  //---------------------------------------------------------------------------------------------------------------
  //---------------------------------------------------------------------------------------------------------------
  E_PROGRESS.PROGRESS_STARTUP:
    _InstanceCtrl[E_INSTANCE.BUFFER_OUTFEED_ROBOT].Cmd   := E_INSTANCE_CMD.DISABLE;
    //-----------------------------------------------------------------------------------
    CASE _InstanceState[E_INSTANCE.BUFFER_OUTFEED_ROBOT].State
    OF
      E_INSTANCE_STATE.DISABLED:
        CASE _InstanceState[E_INSTANCE.BUFFER_OUTFEED_ROBOT].Progress
        OF
          E_PROGRESS.PROGRESS_BUSY:           // check for startup to be done
          _eState                                 := E_PROGRESS.PROGRESS_CHECK; // go check next insatnce
        END_CASE
    END_CASE

  //---------------------------------------------------------------------------------------------------------------
  //---------------------------------------------------------------------------------------------------------------
  E_PROGRESS.PROGRESS_CHECK:
    _InstanceCtrl[E_INSTANCE.OUTFEED_ROBOT_R1].Cmd   := E_INSTANCE_CMD.DISABLE;
    //-----------------------------------------------------------------------------------
    CASE _InstanceState[E_INSTANCE.OUTFEED_ROBOT_R1].State
    OF
      E_INSTANCE_STATE.DISABLED:
        CASE _InstanceState[E_INSTANCE.OUTFEED_ROBOT_R1].Progress
        OF
          E_PROGRESS.PROGRESS_BUSY:           // check for startup to be done
          _eState                                 := E_PROGRESS.PROGRESS_OCCUPIED; // go check next insatnce
        END_CASE
    END_CASE

  //---------------------------------------------------------------------------------------------------------------
  //---------------------------------------------------------------------------------------------------------------
  E_PROGRESS.PROGRESS_OCCUPIED:
    _InstanceCtrl[E_INSTANCE.OUTFEED_ROBOT_R2].Cmd   := E_INSTANCE_CMD.DISABLE;
    //-----------------------------------------------------------------------------------
    CASE _InstanceState[E_INSTANCE.OUTFEED_ROBOT_R2].State
    OF
      E_INSTANCE_STATE.DISABLED:
        CASE _InstanceState[E_INSTANCE.OUTFEED_ROBOT_R2].Progress
        OF
          E_PROGRESS.PROGRESS_BUSY:           // check for startup to be done
          _eState                                 := E_PROGRESS.PROGRESS_WORKING; // go check next insatnce
        END_CASE
    END_CASE

  //---------------------------------------------------------------------------------------------------------------
  //---------------------------------------------------------------------------------------------------------------
  E_PROGRESS.PROGRESS_WORKING:
    _InstanceCtrl[E_INSTANCE.SENDER_FAST].Cmd     := E_INSTANCE_CMD.DISABLE;
    //-----------------------------------------------------------------------------------
    CASE _InstanceState[E_INSTANCE.SENDER_FAST].State
    OF
      E_INSTANCE_STATE.DISABLED:
        CASE _InstanceState[E_INSTANCE.SENDER_FAST].Progress
        OF
          E_PROGRESS.PROGRESS_BUSY:           // check for startup to be done
          _eState                                 := E_PROGRESS.PROGRESS_STILL_WORKING; // go check next insatnce
        END_CASE
    END_CASE

  //---------------------------------------------------------------------------------------------------------------
  //---------------------------------------------------------------------------------------------------------------
  E_PROGRESS.PROGRESS_STILL_WORKING:
    _InstanceCtrl[E_INSTANCE.SENDER_BUFFER_INFEED].Cmd   := E_INSTANCE_CMD.DISABLE;
    //-----------------------------------------------------------------------------------
    CASE _InstanceState[E_INSTANCE.SENDER_BUFFER_INFEED].State
    OF
      E_INSTANCE_STATE.DISABLED:
        CASE _InstanceState[E_INSTANCE.SENDER_BUFFER_INFEED].Progress
        OF
          E_PROGRESS.PROGRESS_BUSY:           // check for startup to be done
          _eState                                 := E_PROGRESS.PROGRESS_DONE;
        END_CASE
    END_CASE
END_CASE
//-----------------------------------------------------------------------------
//-----------------------------------------------------------------------------

Init                                              := _eState;
END_METHOD

PROPERTY InstanceCtrl : REFERENCE TO ARRAY[1..MAX_PROCESS] OF ST_INSTANCE_CTRL
SET
_InstanceCtrl REF= InstanceCtrl;
END_SET
END_PROPERTY

PROPERTY InstanceState : REFERENCE TO ARRAY[1..MAX_PROCESS] OF ST_INSTANCE_STATE
SET
_InstanceState REF= InstanceState;
END_SET
END_PROPERTY

METHOD ListData   : E_PROGRESS  // simulates data entry from transfersystem into BUFFER_INFEED linked list
VAR_INPUT
  Start           : BOOL;
  Reset           : BOOL;
END_VAR
VAR_INST
  _nBit,
  _nExp           : BYTE;
  _nMod           : UINT := 5;
  _nCount         : UINT;
  _eStateProgress : E_PROGRESS;

  _ProcessData    : ST_PROCESS_DATA;
  _Rslt           : ST_PROCESS_LIST_RESULT;

  _nMinListCount  : UDINT := 1;
  _nWaitcountLast,
  _nWaitCount     : UDINT;

  _tMsg           : ST_Message;
  _eMessageLevel  : E_MessageType;  // manual local switch for enabling info messages
END_VAR
IF Reset
THEN
  _nCount                     := 1;
  _eStateProgress             := E_PROGRESS.PROGRESS_INIT;
  _ItfProcessList[E_INSTANCE.BUFFER_INFEED].InitList();
END_IF

_tMsg.eDevice                 := _stMsg.eDevice; 

CASE _eStateProgress
OF
   E_PROGRESS.PROGRESS_INIT:
    IF Start
    THEN
      _eStateProgress         :=  E_PROGRESS.PROGRESS_BUSY;
    END_IF

  E_PROGRESS.PROGRESS_BUSY:
    CASE _nLoadCase
    OF
      0:  // fully loaded
        _eStateProgress       := E_PROGRESS.PROGRESS_CHECK;
        _nLoadCaseOld         := _nLoadCase;

        IF (_eMessageLevel > E_MessageType.eMessageError)
        THEN
          _tMsg.eType          := E_MessageType.eMessageInfo;
          _tMsg.eSubdevice     := e_Subdevice.Application;
          _tMsg.iErrorNumber   := _nLoadCase;
          _tMsg.sText          := concat(TO_STRING(_eState), ': ListData');
          f_MessageSet(_stMsg);
        END_IF


      1:  // static bits
        _eStateProgress       := E_PROGRESS.PROGRESS_PREPARE;
        _nLoadCaseOld         := _nLoadCase;

        IF (_eMessageLevel > E_MessageType.eMessageError)
        THEN
          _tMsg.eType          := E_MessageType.eMessageInfo;
          _tMsg.eSubdevice     := e_Subdevice.Application;
          _tMsg.iErrorNumber   := _nLoadCase;
          _tMsg.sText          := concat(TO_STRING(_eState), ': ListData');
          f_MessageSet(_stMsg);
        END_IF


      2:  // incrementing bits
        _eStateProgress       := E_PROGRESS.PROGRESS_STARTUP;
        _nLoadCaseOld         := _nLoadCase;

        IF (_eMessageLevel > E_MessageType.eMessageError)
        THEN
          _tMsg.eType          := E_MessageType.eMessageInfo;
          _tMsg.eSubdevice     := e_Subdevice.Application;
          _tMsg.iErrorNumber   := _nLoadCase;
          _tMsg.sText          := concat(TO_STRING(_eState), ': ListData');
          f_MessageSet(_stMsg);
        END_IF


      99:
        _eStateProgress       := E_PROGRESS.PROGRESS_WORKING;
        _ProcessData.wTarget  := 0;

        IF (_eMessageLevel > E_MessageType.eMessageError)
        THEN
          _tMsg.eType          := E_MessageType.eMessageInfo;
          _tMsg.eSubdevice     := e_Subdevice.Application;
          _tMsg.iErrorNumber   := _nLoadCase;
          _tMsg.sText          := concat(TO_STRING(_eState), ': _ProcessData.wTarget: ');
          _tMsg.sText          := concat(_stMsg.sText, _ItfProcessCollector[E_INSTANCE.BUFFER_INFEED].BitsToString(_ProcessData.wTarget));
          f_MessageSet(_stMsg);
        END_IF
        _nLoadCase            := _nLoadCaseOld;

    ELSE
        _eStateProgress       := E_PROGRESS.PROGRESS_STARTUP;
    END_CASE
    _nWaitCount               := 0; 
END_CASE
CASE _eStateProgress
OF
  E_PROGRESS.PROGRESS_PREPARE:
    _eStateProgress           := E_PROGRESS.PROGRESS_WORKING;
    _nExp                     := TO_BYTE(ItfProcessCollector[E_INSTANCE.INFEED].StationCount);
    _ProcessData.wTarget      := _ItfProcessCollector[E_INSTANCE.BUFFER_INFEED].To_T_Process(_nExp);

    IF (_nCount MOD _nMod = 0)
    THEN
      _nBit                   := SEL((_nBit>_nExp), _nBit+1, 0);
      _ProcessData.wTarget    := _ItfProcessCollector[E_INSTANCE.BUFFER_INFEED].DelBit(_ProcessData.wTarget, _nBit);
    END_IF
    IF (_nCount MOD (8) = 0)
    THEN
      _nBit                   := 1;
      _ProcessData.wTarget    := _ItfProcessCollector[E_INSTANCE.BUFFER_INFEED].DelBit(_ProcessData.wTarget, _nBit);
    END_IF
    IF (_nCount MOD (16) = 0)
    THEN
      _nBit                   := 2;
      _ProcessData.wTarget    := _ItfProcessCollector[E_INSTANCE.BUFFER_INFEED].DelBit(_ProcessData.wTarget, _nBit);
    END_IF
    IF (_nCount MOD (24) = 0)
    THEN
      _nBit                   := 3;
      _ProcessData.wTarget    := _ItfProcessCollector[E_INSTANCE.BUFFER_INFEED].DelBit(_ProcessData.wTarget, _nBit);
    END_IF
    IF (_nCount MOD (32) = 0)
    THEN
      _nBit                   := 4;
      _ProcessData.wTarget    := _ItfProcessCollector[E_INSTANCE.BUFFER_INFEED].DelBit(_ProcessData.wTarget, _nBit);
    END_IF
    IF (_nCount MOD (40) = 0)
    THEN
      _nBit                   := 5;
      _ProcessData.wTarget    := _ItfProcessCollector[E_INSTANCE.BUFFER_INFEED].DelBit(_ProcessData.wTarget, _nBit);
    END_IF
    IF (_nCount MOD (48) = 0)
    THEN
      _nBit                   := 6;
      _ProcessData.wTarget    := _ItfProcessCollector[E_INSTANCE.BUFFER_INFEED].DelBit(_ProcessData.wTarget, _nBit);
    END_IF
    IF (_nCount MOD (60) = 0)
    THEN
      _nBit                   := 7;
      _ProcessData.wTarget    := _ItfProcessCollector[E_INSTANCE.BUFFER_INFEED].DelBit(_ProcessData.wTarget, _nBit);
    END_IF
    IF (_nCount MOD (72) = 0)
    THEN
      _nBit                   := 8;
      _ProcessData.wTarget    := _ItfProcessCollector[E_INSTANCE.BUFFER_INFEED].DelBit(_ProcessData.wTarget, _nBit);
    END_IF
    IF (_nCount MOD (84) = 0)
    THEN
      _nBit                   := 9;
      _ProcessData.wTarget    := _ItfProcessCollector[E_INSTANCE.BUFFER_INFEED].DelBit(_ProcessData.wTarget, _nBit);
    END_IF
    IF (_nCount MOD (96) = 0)
    THEN
      _nBit                   := 10;
      _ProcessData.wTarget    := _ItfProcessCollector[E_INSTANCE.BUFFER_INFEED].DelBit(_ProcessData.wTarget, _nBit);
    END_IF
    IF (_nCount MOD (108) = 0)
    THEN
      _nBit                   := 11;
      _ProcessData.wTarget    := _ItfProcessCollector[E_INSTANCE.BUFFER_INFEED].DelBit(_ProcessData.wTarget, _nBit);
    END_IF
END_CASE
CASE _eStateProgress
OF
  E_PROGRESS.PROGRESS_STARTUP:
    _eStateProgress           := E_PROGRESS.PROGRESS_WORKING;
    _nExp                     := TO_BYTE(ItfProcessCollector[E_INSTANCE.INFEED].StationCount);
    _ProcessData.wTarget      := _ItfProcessCollector[E_INSTANCE.BUFFER_INFEED].To_T_Process(_nExp);

    IF (_nCount MOD _nMod = 0)
    THEN
      _nBit                   := SEL((_nBit>_nExp), _nBit+1, 0);
      _ProcessData.wTarget    := _ItfProcessCollector[E_INSTANCE.BUFFER_INFEED].DelBit(_ProcessData.wTarget, _nBit);
    END_IF
(*
    IF (_nCount MOD (8) = 0)
    THEN
      _nBit                   := SEL((_nBit>_nExp), _nBit+1, 0);
      _ProcessData.wTarget    := _ItfProcessCollector[E_INSTANCE.BUFFER_INFEED].DelBit(_ProcessData.wTarget, _nBit);
    END_IF
    IF (_nCount MOD (16) = 0)
    THEN
      _nBit                   := SEL((_nBit>_nExp), _nBit+1, 0);
      _ProcessData.wTarget    := _ItfProcessCollector[E_INSTANCE.BUFFER_INFEED].DelBit(_ProcessData.wTarget, _nBit);
    END_IF
    IF (_nCount MOD (24) = 0)
    THEN
      _nBit                   := SEL((_nBit>_nExp), _nBit+1, 0);
      _ProcessData.wTarget    := _ItfProcessCollector[E_INSTANCE.BUFFER_INFEED].DelBit(_ProcessData.wTarget, _nBit);
    END_IF
    IF (_nCount MOD (32) = 0)
    THEN
      _nBit                   := SEL((_nBit>_nExp), _nBit+1, 0);
      _ProcessData.wTarget    := _ItfProcessCollector[E_INSTANCE.BUFFER_INFEED].DelBit(_ProcessData.wTarget, _nBit);
    END_IF
    IF (_nCount MOD (40) = 0)
    THEN
      _nBit                   := SEL((_nBit>_nExp), _nBit+1, 0);
      _ProcessData.wTarget    := _ItfProcessCollector[E_INSTANCE.BUFFER_INFEED].DelBit(_ProcessData.wTarget, _nBit);
    END_IF
    IF (_nCount MOD (48) = 0)
    THEN
      _nBit                   := SEL((_nBit>_nExp), _nBit+1, 0);
      _ProcessData.wTarget    := _ItfProcessCollector[E_INSTANCE.BUFFER_INFEED].DelBit(_ProcessData.wTarget, _nBit);
    END_IF
*)
END_CASE
CASE _eStateProgress
OF
  E_PROGRESS.PROGRESS_CHECK:
    _eStateProgress           := E_PROGRESS.PROGRESS_WORKING;
    _nExp                     := TO_BYTE(ItfProcessCollector[E_INSTANCE.INFEED].StationCount);
    _ProcessData.wTarget      := _ItfProcessCollector[E_INSTANCE.BUFFER_INFEED].To_T_Process(_nExp);

    IF (_eMessageLevel > E_MessageType.eMessageError)
    THEN
      _tMsg.eType            := E_MessageType.eMessageInfo;
      _tMsg.eSubdevice       := e_Subdevice.Application;
      _tMsg.iErrorNumber     := _nLoadCase;
      _tMsg.sText            := concat(TO_STRING(_eState), ': _ProcessData.wTarget: ');
      _tMsg.sText            := concat(_stMsg.sText, _ItfProcessCollector[E_INSTANCE.BUFFER_INFEED].BitsToString(_ProcessData.wTarget));
      f_MessageSet(_stMsg);
    END_IF
END_CASE
CASE _eStateProgress
OF
  E_PROGRESS.PROGRESS_WORKING:
    _Rslt                     := _ItfProcessList[E_INSTANCE.BUFFER_INFEED].AddTailValue(_ProcessData);

    IF (_Rslt.wState = 0)
    THEN
      _nCount                 := _nCount + 1;
      _eStateProgress         := E_PROGRESS.PROGRESS_OCCUPIED;
    ELSE
      _eStateProgress         := E_PROGRESS.PROGRESS_ERROR;
    END_IF
END_CASE
CASE _eStateProgress
OF
  E_PROGRESS.PROGRESS_OCCUPIED:
    _nWaitCount               := _nWaitCount + 1;

    IF (_ItfProcessList[E_INSTANCE.BUFFER_INFEED].Count < _nMinListCount)
    THEN
      _nWaitCountLast         := _nWaitCount;
      _eStateProgress         :=  E_PROGRESS.PROGRESS_INIT;
    END_IF
END_CASE

ListData                      := _eStateProgress;
END_METHOD

PROPERTY MessageLevel : e_MessageType
GET
MessageLevel := _MessageLevel;
END_GET
SET
_MessageLevel := MessageLevel;
END_SET
END_PROPERTY

METHOD Proceed : E_PROGRESS
VAR_INPUT
  Execute     : BOOL;
END_VAR
VAR_INST
  _nErrorId               : UDINT;
  _eState                 : E_PROGRESS;

  _nExp                   : BYTE;
  _WriteData              : ST_PROCESS_DATA;
  _WriteResult            : ST_PROCESS_LIST_RESULT;

  _eInst                  : E_INSTANCE;
  _TransportState         : E_XTS_TRANSPORT_STATE;
  _bDbg : BOOL;
END_VAR
//-----------------------------------------------------------------------------
IF NOT Execute 
THEN 
	_eState                       := E_PROGRESS.PROGRESS_INIT; 
END_IF 
//-----------------------------------------------------------------------------
IF NOT Check() 
THEN 
	Proceed                       := E_PROGRESS.PROGRESS_ERROR; 
	RETURN; 
END_IF
//-----------------------------------------------------------------------------
//-----------------------------------------------------------------------------
CASE _eState
OF
  E_PROGRESS.PROGRESS_INIT:
    IF Execute
    THEN
      _nErrorId                 := 0;

      IF (_XtsTransportState.GroupInfo.AxisCountEnabled = MAX_MOVER) AND
         (_XtsTransportState.GroupInfo.AxisCount        = MAX_MOVER)
      THEN
        _eState                 := E_PROGRESS.PROGRESS_BUSY;
        _XtsTransportCtrl.Cmd   := E_XTS_TRANSPORT_CTRL.CMD_NULL;

        IF (_MessageLevel > E_MessageType.eMessageError)
        THEN
          _stMsg.eType          := E_MessageType.eMessageInfo;
          _stMsg.eSubdevice     := e_Subdevice.Application_Proceed;
          _stMsg.iErrorNumber   := 0;
          _stMsg.sText          := concat(TO_STRING(_eState), ': ');
          f_MessageSet(_stMsg);
        END_IF
      ELSE
        _nErrorId               := _eState;

        _eState                 := E_PROGRESS.PROGRESS_ERROR;

        _stMsg.eType            := E_MessageType.eMessageError;
        _stMsg.eSubdevice       := e_Subdevice.Application_Proceed;
        _stMsg.iErrorNumber     := _nErrorId;
        _stMsg.sText            := concat(TO_STRING(_eState), ': ');
        _stMsg.sText            := concat(_stMsg.sText, TO_STRING(_XtsTransportState.GroupInfo.AxisCountEnabled));
        _stMsg.sText            := concat(_stMsg.sText, ' / ');
        _stMsg.sText            := concat(_stMsg.sText, TO_STRING(_XtsTransportState.GroupInfo.AxisCount));
        _stMsg.sText            := concat(_stMsg.sText, ' CaGroup Axis mismatch');
        f_MessageSet(_stMsg);
      END_IF
    END_IF


  E_PROGRESS.PROGRESS_BUSY:
    _XtsTransportCtrl.Cmd       := E_XTS_TRANSPORT_CTRL.CMD_TRANSPORT_RESTART;

    IF (_XtsTransportState.State = E_XTS_TRANSPORT_STATE.TRANSPORT_RESTART + E_PROGRESS.PROGRESS_ERROR)
    THEN
      _eState                   := E_PROGRESS.PROGRESS_ERROR;
      _TransportState           := _XtsTransportState.State MOD E_PROGRESS.PROGRESS_ERROR;

      _stMsg.eType              := E_MessageType.eMessageError;
      _stMsg.eSubdevice         := e_Subdevice.Application_Proceed;
      _stMsg.iErrorNumber       := _nErrorId;
      _stMsg.sText              := concat(TO_STRING(_eState), ': ');
      _stMsg.sText              := concat(_stMsg.sText, TO_STRING(_TransportState));
      f_MessageSet(_stMsg);

    ELSIF (_XtsTransportState.State = E_XTS_TRANSPORT_STATE.TRANSPORT_RESTART + E_PROGRESS.PROGRESS_DONE)
    THEN
      _eState                   := E_PROGRESS.PROGRESS_WORKING;
      _TransportState           := _XtsTransportState.State MOD E_PROGRESS.PROGRESS_DONE;

      IF (_MessageLevel > E_MessageType.eMessageError)
      THEN
        _stMsg.eType            := E_MessageType.eMessageInfo;
        _stMsg.eSubdevice       := e_Subdevice.Application_Proceed;
        _stMsg.iErrorNumber     := 0;
        _stMsg.sText            := concat(TO_STRING(_eState), ': ');
        _stMsg.sText            := concat(_stMsg.sText, TO_STRING(_TransportState));
        f_MessageSet(_stMsg);
      END_IF
    END_IF

END_CASE
//-----------------------------------------------------------------------------
//-----------------------------------------------------------------------------
CASE _eState
OF
  E_PROGRESS.PROGRESS_WORKING:
    ListData(TRUE, FALSE);    // start writing linked list entries into BUFFER_INFEED

    FOR _eInst := E_INSTANCE.BUFFER_INFEED TO E_INSTANCE.SENDER_BUFFER_INFEED
    DO
      // handshakes to instances: 
      // - deconstruct this for your own implementation
      CASE _InstanceState[_eInst].State
      OF
        E_INSTANCE_STATE.DISABLED:
          CASE _InstanceState[_eInst].Progress
          OF
            E_PROGRESS.PROGRESS_BUSY:
              _InstanceCtrl[_eInst].Cmd    := E_INSTANCE_CMD.ENABLE;
          END_CASE
      
        E_INSTANCE_STATE.ENABLED:
          CASE _InstanceState[_eInst].Progress
          OF
            E_PROGRESS.PROGRESS_OCCUPIED:
              _InstanceCtrl[_eInst].Cmd    := E_INSTANCE_CMD.PROCEED;
          END_CASE
      
        E_INSTANCE_STATE.WORKING:
          CASE _InstanceState[_eInst].Progress
          OF
            E_PROGRESS.PROGRESS_BUSY:
              _tonProcess [_eInst]
                              (IN         := FALSE, 
                               PT         := _tProcess[_eInst]);

              IF (_eInst > E_INSTANCE.OUTFEED_ROBOT_R2) OR
                 (_eInst < E_INSTANCE.OUTFEED_ROBOT_R1)
              THEN
                _InstanceCtrl[_eInst].Cmd   := E_INSTANCE_CMD.WORK;
              ELSE
                IF (_InstanceState[E_INSTANCE.OUTFEED_ROBOT_R1].State = 
                    _InstanceState[E_INSTANCE.OUTFEED_ROBOT_R2].State )
                THEN
                  // in this example the outfeed instances are working in sync
                  _InstanceCtrl[_eInst].Cmd := E_INSTANCE_CMD.WORK;
                ELSE
                  CASE _InstanceState[E_INSTANCE.OUTFEED_ROBOT_R2].State
                  OF
                    E_INSTANCE_STATE.ENABLED:
                      // in case R2 is empty --> unload R1
                      _InstanceCtrl[E_INSTANCE.OUTFEED_ROBOT_R1].Cmd := E_INSTANCE_CMD.WORK;
                  END_CASE
                END_IF
              END_IF
      
      
            E_PROGRESS.PROGRESS_CHECK:
              _tonProcess [_eInst]
                              (IN         := TRUE, 
                               PT         := _tProcess[_eInst]);
      
              IF _tonProcess [_eInst].Q
              THEN
                _InstanceCtrl[_eInst].Cmd := E_INSTANCE_CMD.FINISH;
              END_IF
          END_CASE


        E_INSTANCE_STATE.FINISH:
          CASE _InstanceState[_eInst].Progress
          OF
            E_PROGRESS.PROGRESS_BUSY:
              _InstanceCtrl[_eInst].Cmd    := E_INSTANCE_CMD.FINISH;

            E_PROGRESS.PROGRESS_OCCUPIED:
              _InstanceCtrl[_eInst].Cmd    := E_INSTANCE_CMD.PROCEED;
          END_CASE
        END_CASE
    END_FOR
END_CASE
//-----------------------------------------------------------------------------
//-----------------------------------------------------------------------------

Proceed                            := _eState;
END_METHOD

PROPERTY ProcessLinkedLists : REFERENCE TO ARRAY[1..MAX_PROCESS] OF I_Process_LinkedList
SET
_ItfProcessList REF= ProcessLinkedLists;
END_SET
END_PROPERTY

PROPERTY State : REFERENCE TO ST_APP_STATE
SET
_State ref= State;
END_SET
END_PROPERTY

METHOD Work : E_PROGRESS  // cyclic handshakes with timers, 
                          // this procedure you have to build for your own application. 
                          // This simulated work method is here 
                          // because it was convinient for me to do so
VAR_INPUT
  Execute                 : BOOL;
END_VAR
VAR_INST
  _nErrorId               : UDINT;
  _eRslt,
  _eState                 : E_PROGRESS;

  _nExp                   : BYTE;
  _WriteData              : ST_PROCESS_DATA;
  _WriteResult            : ST_PROCESS_LIST_RESULT;

  _eInst                  : E_INSTANCE;
  _bDbg : BOOL;

  _TransportState         : E_XTS_TRANSPORT_STATE;
  _JobResult              : E_PROGRESS;
END_VAR
//-----------------------------------------------------------------------------
IF NOT Execute 
THEN 
	_eState                       := E_PROGRESS.PROGRESS_INIT; 
END_IF 
//-----------------------------------------------------------------------------
IF NOT Check() 
THEN 
	Work                          := E_PROGRESS.PROGRESS_ERROR; 
	RETURN; 
END_IF
//-----------------------------------------------------------------------------
//-----------------------------------------------------------------------------
CASE _eState
OF
  E_PROGRESS.PROGRESS_INIT:
    IF Execute
    THEN
      _nErrorId                 := 0;

      IF (_XtsTransportState.GroupInfo.AxisCountEnabled = MAX_MOVER) AND
         (_XtsTransportState.GroupInfo.AxisCount        = MAX_MOVER)
      THEN
        _eState                 := E_PROGRESS.PROGRESS_BUSY;
        _XtsTransportCtrl.Cmd   := E_XTS_TRANSPORT_CTRL.CMD_NULL;
        _eRslt                  := Clear(FALSE);

        IF (_MessageLevel > E_MessageType.eMessageError)
        THEN
          _stMsg.eType          := E_MessageType.eMessageInfo;
          _stMsg.eSubdevice     := e_Subdevice.Application_Work;
          _stMsg.iErrorNumber   := 0;
          _stMsg.sText          := concat(TO_STRING(_eState), ': ');
          f_MessageSet(_stMsg);
        END_IF
      ELSE
        _nErrorId               := _XtsTransportState.GroupInfo.AxisCountEnabled;
        _eState                 := E_PROGRESS.PROGRESS_ERROR;

        _stMsg.eType            := E_MessageType.eMessageError;
        _stMsg.eSubdevice       := e_Subdevice.Application_Work;
        _stMsg.iErrorNumber     := _nErrorId;
        _stMsg.sText            := concat(TO_STRING(_eState), ': ');
        _stMsg.sText            := concat(_stMsg.sText, TO_STRING(_XtsTransportState.GroupInfo.AxisCountEnabled));
        _stMsg.sText            := concat(_stMsg.sText, ' / ');
        _stMsg.sText            := concat(_stMsg.sText, TO_STRING(_XtsTransportState.GroupInfo.AxisCount));
        _stMsg.sText            := concat(_stMsg.sText, ' CaGroup Axis mismatch');
        f_MessageSet(_stMsg);
      END_IF
    END_IF


  E_PROGRESS.PROGRESS_BUSY:
    _eRslt                      := Clear(TRUE);

    IF (_eRslt = E_PROGRESS.PROGRESS_DONE)
    THEN
      _XtsTransportCtrl.Cmd     := E_XTS_TRANSPORT_CTRL.CMD_TRANSPORT_START;
  
      IF (_XtsTransportState.State = E_XTS_TRANSPORT_STATE.TRANSPORT_START + E_PROGRESS.PROGRESS_ERROR)
      THEN
        _eState                 := E_PROGRESS.PROGRESS_ERROR;
        _TransportState         := _XtsTransportState.State MOD E_PROGRESS.PROGRESS_ERROR;

        _stMsg.eType            := E_MessageType.eMessageError;
        _stMsg.eSubdevice       := e_Subdevice.Application_Work;
        _stMsg.iErrorNumber     := _nErrorId;
        _stMsg.sText            := concat(TO_STRING(_eState), ': ');
        _stMsg.sText            := concat(_stMsg.sText, TO_STRING(_TransportState));
        f_MessageSet(_stMsg);
  
      ELSIF (_XtsTransportState.State = E_XTS_TRANSPORT_STATE.TRANSPORT_START + E_PROGRESS.PROGRESS_DONE)
      THEN
        _eState                 := E_PROGRESS.PROGRESS_PREPARE;
        _TransportState         := _XtsTransportState.State MOD E_PROGRESS.PROGRESS_DONE;

        IF (_MessageLevel > E_MessageType.eMessageError)
        THEN
          _stMsg.eType          := E_MessageType.eMessageInfo;
          _stMsg.eSubdevice     := e_Subdevice.Application_Work;
          _stMsg.iErrorNumber   := 0;
          _stMsg.sText          := concat(TO_STRING(_eState), ': ');
          _stMsg.sText          := concat(_stMsg.sText, TO_STRING(_TransportState));
          f_MessageSet(_stMsg);
        END_IF
      END_IF
    END_IF
END_CASE
//-----------------------------------------------------------------------------
//-----------------------------------------------------------------------------
CASE _eState
OF
  E_PROGRESS.PROGRESS_PREPARE:  // SENDER_BUFFER_INFEED sends the first batch of movers to BUFFER_INFEED
                                //  - after sending the first batch 
                                //    --> the transfersystem (ListData) may start writing entries into BUFFER_INFEED
    CASE _InstanceState[E_INSTANCE.SENDER_BUFFER_INFEED].State
    OF
    E_INSTANCE_STATE.DISABLED:

      CASE _InstanceState[E_INSTANCE.SENDER_BUFFER_INFEED].Progress
      OF
      E_PROGRESS.PROGRESS_BUSY:
        _nExp                   := TO_BYTE(ItfProcessCollector[E_INSTANCE.INFEED].StationCount);
        _WriteData.wTarget      := _ItfProcessCollector[E_INSTANCE.SENDER_BUFFER_INFEED].To_T_Process(_nExp);

        _WriteResult            := _ItfProcessList[E_INSTANCE.SENDER_BUFFER_INFEED].AddTailValue(_WriteData);

        IF (_WriteResult.wState <> 0)
        THEN
          _eState               := E_PROGRESS.PROGRESS_ERROR;

          _stMsg.eType          := E_MessageType.eMessageError;
          _stMsg.eSubdevice     := e_Subdevice.Application_Work;
          _stMsg.iErrorNumber   := _WriteResult.wState;
          _stMsg.sText          := concat(TO_STRING(_eState), ': ');
          _stMsg.sText          := concat(_stMsg.sText, TO_STRING(e_Subdevice.Process_LinkedList_AddTail));
          f_MessageSet(_stMsg);

        ELSE
          ListData(FALSE, TRUE);    // init linked list from simulated transfersystem (timer based entry into linked list)
          _eState               := E_PROGRESS.PROGRESS_CHECK;

          IF (_MessageLevel > E_MessageType.eMessageError)
          THEN
            _stMsg.eType        := E_MessageType.eMessageInfo;
            _stMsg.eSubdevice   := e_Subdevice.Application_Work;
            _stMsg.iErrorNumber := 0;
            _stMsg.sText        := concat(TO_STRING(_eState), ': ');
            _stMsg.sText        := concat(_stMsg.sText, TO_STRING(e_Subdevice.Process_LinkedList_AddTail));
            f_MessageSet(_stMsg);
          END_IF
        END_IF
      END_CASE
    END_CASE
END_CASE
//-----------------------------------------------------------------------------
//-----------------------------------------------------------------------------
CASE _eState
OF
  E_PROGRESS.PROGRESS_CHECK:
    _eState := E_PROGRESS.PROGRESS_OCCUPIED; 
END_CASE
//-----------------------------------------------------------------------------
//-----------------------------------------------------------------------------
CASE _eState
OF
  E_PROGRESS.PROGRESS_OCCUPIED:
    _eState := E_PROGRESS.PROGRESS_WORKING;

    IF (_MessageLevel > E_MessageType.eMessageError)
    THEN
      _stMsg.eType            := E_MessageType.eMessageInfo;
      _stMsg.eSubdevice       := e_Subdevice.Application_Work;
      _stMsg.iErrorNumber     := 0;
      _stMsg.sText            := concat(TO_STRING(_eState), ': ');
      f_MessageSet(_stMsg);
    END_IF
END_CASE
//-----------------------------------------------------------------------------
//-----------------------------------------------------------------------------
CASE _eState
OF
  E_PROGRESS.PROGRESS_WORKING:
    ListData(TRUE, FALSE);    // start writing linked list entries into BUFFER_INFEED

    FOR _eInst := E_INSTANCE.BUFFER_INFEED TO E_INSTANCE.SENDER_BUFFER_INFEED
    DO
      // handshakes to instances: 
      // - deconstruct this for your own implementation
      CASE _InstanceState[_eInst].State
      OF
        E_INSTANCE_STATE.DISABLED:
          CASE _InstanceState[_eInst].Progress
          OF
            E_PROGRESS.PROGRESS_BUSY:
              _InstanceCtrl[_eInst].Cmd    := E_INSTANCE_CMD.ENABLE;
          END_CASE
      
        E_INSTANCE_STATE.ENABLED:
          CASE _InstanceState[_eInst].Progress
          OF
            E_PROGRESS.PROGRESS_OCCUPIED:
              _InstanceCtrl[_eInst].Cmd    := E_INSTANCE_CMD.PROCEED;
          END_CASE

        E_INSTANCE_STATE.WORKING:
          CASE _InstanceState[_eInst].Progress
          OF
            E_PROGRESS.PROGRESS_BUSY:
              _tonProcess [_eInst]
                              (IN         := FALSE, 
                               PT         := _tProcess[_eInst]);

              IF (_eInst > E_INSTANCE.OUTFEED_ROBOT_R2) OR
                 (_eInst < E_INSTANCE.OUTFEED_ROBOT_R1) OR
                 (_bSingleOutput)
              THEN
                _InstanceCtrl[_eInst].Cmd   := E_INSTANCE_CMD.WORK;
              ELSE
                IF (_InstanceState[E_INSTANCE.OUTFEED_ROBOT_R1].State = 
                    _InstanceState[E_INSTANCE.OUTFEED_ROBOT_R2].State )
                THEN
                  // in this example the outfeed instances are working in sync
                  _InstanceCtrl[_eInst].Cmd := E_INSTANCE_CMD.WORK;
                END_IF
              END_IF
      
      
            E_PROGRESS.PROGRESS_CHECK:
              _tonProcess [_eInst]
                              (IN         := TRUE, 
                               PT         := _tProcess[_eInst]);
      
              IF _tonProcess [_eInst].Q
              THEN
                _InstanceCtrl[_eInst].Cmd := E_INSTANCE_CMD.FINISH;
              END_IF
          END_CASE


        E_INSTANCE_STATE.FINISH:
          CASE _InstanceState[_eInst].Progress
          OF
            E_PROGRESS.PROGRESS_BUSY:
              _tonProcess [_eInst]
                              (IN         := FALSE, 
                               PT         := _tProcess[_eInst]);

              _InstanceCtrl[_eInst].Cmd    := E_INSTANCE_CMD.FINISH;

            E_PROGRESS.PROGRESS_OCCUPIED:
              _InstanceCtrl[_eInst].Cmd    := E_INSTANCE_CMD.PROCEED;
          END_CASE
        END_CASE
    END_FOR
END_CASE
//-----------------------------------------------------------------------------
//-----------------------------------------------------------------------------

Work                            := _eState;
END_METHOD

PROPERTY XtsTransportCtrl : REFERENCE TO ST_XTS_TRANSPORT_CTRL
SET
_XtsTransportCtrl REF= XtsTransportCtrl;
END_SET
END_PROPERTY

PROPERTY XtsTransportState : REFERENCE TO ST_XTS_TRANSPORT_STATE
SET
_XtsTransportState REF= XtsTransportState;
END_SET
END_PROPERTY

END_FUNCTION_BLOCK

// ---- APPLICATION/_types/Instance/fb_Instance.TcPOU
//---------------------------------------------------------------------------------------------------------------
//
//  HAUD 2024.11.21
//
//
//  fb_Instance
//-----------------------------------------------------------------------------
//  - base class for my process instance to work with fb_ProcessCollector
//
//  - _nProcess --> whoami, this is me
//
//  - fb_ProcessCollector[_nProcess].Cycle() is called in APPLICATION(PRG)
//    - handles range of XtsStations
//    - range must be closed and in consecutive order
//
//    - combines states into bitmasks, one bit per XtsStation
//    - controls forwarding of commands to range of XtsStations 
//      (see fb_ProcessCollector.Cycle())
//
//  - reference to all _ItfProcessCollector(I_ProcessCollector)[]
//    - _ItfProcessCollector[nProcess] Get/Set properties and methods
//
//  - Control / State of my process
//    - datafield for control and state provided
//    - _Ctrl 
//      --> commands to my process; fb_ProcessCollector[_nProcess]
//      --> is linked (REF=) automatically in Check()
//
//      Cmd               : E_PROCESS_CTRL; // command enum for my process
//      ProcessTarget     : UINT;           // target of my process
//      ActivateStation   : WORD;           // is checked for every job
//                                          // every bit is a XtsStation
//
//      NestMask          : BYTE;           // one mask for all XtsStations
//      - every bit is a PosStop in a XtsStation
//      - copied to every XtsStation in my process when movers are about to leave
//
//    - _State
//      --> satus information from my process
//      --> check for plausible StationLast / StationFirst range of XtsStations
//
//      State             : E_PROCESS_STATE;  // state enuum from my process
//      Result            : E_PROGRESS;       // substate from my process, BUSY signals state is ready for interaction
//      Check             : E_PROCESS_CHECK;  // plausibility check of StationLast and StationFirst 
//
//
//  - basic check and var names, so you can build your procedures with it
//
//  - processes may be connected via linked list, you decide.
//    - linked list for processes is intended to work as job buffer
//    - linked list provides information via ST_PROCESS_DATA, 
//      add what you have to in there
//    - linked ist to all process instances provided
//
//  - inherit this base class for your application, call Check() cyclic
//
//---------------------------------------------------------------------------------------------------------------//
// This SOFTWARE is provided as an Exemple by THE PROVIDER "as is" and "with all faults." THE PROVIDER makes no  //
// representations or warranties of any kind concerning the safety, suitability, lack of viruses, inaccuracies,  //
// typographical errors, or other harmful components of this SOFTWARE. There are inherent dangers in the use of  //
// any software, and you are solely responsible for determining whether this SOFTWARE is compatible with your    //
// equipment and other software installed on your equipment. You are also solely responsible for the protection  //
// of your equipment and backup of your data, and THE PROVIDER will not be liable for any damages you may suffer //
// in connection with using, modifying, or distributing this SOFTWARE.                                           //
//---------------------------------------------------------------------------------------------------------------//
FUNCTION_BLOCK fb_Instance
VAR
  // process index
  _nProcess               : E_INSTANCE;           // whoami

  _InstanceCtrl           : REFERENCE TO ARRAY[1..MAX_PROCESS] OF ST_INSTANCE_CTRL;
  _InstanceState          : REFERENCE TO ARRAY[1..MAX_PROCESS] OF ST_INSTANCE_STATE;

  _eCmd,
  _eCmdOld                : E_INSTANCE_CMD;       // commands for local state machine
  _eStateInstance         : E_INSTANCE_STATE;     // local state machine for infeed procedure

  _eResult,
  _eStateProgress         : E_PROGRESS;           // substate for lacal state machine

  _eInit                  : E_PROGRESS;           // startup
  _eCheck                 : E_INSTANCE_CHECK;     // pointer checks


  // local ctrl / state datafields for you to use, connected by reference to _ItfProcessCollector[_nProcess]
  _Ctrl                   : ST_PROCESS_CTRL;      // control to write, connected by reference to _ItfProcessCollector
  _State                  : ST_PROCESS_STATE;     // state   to read,  connected by reference to _ItfProcessCollector

  _ItfProcessCollector    : ARRAY[1..MAX_PROCESS] OF I_ProcessCollector;    // information and configuration of the connected ProcessCollector for given range of XtsStations

  _ItfProcessList         : ARRAY[1..MAX_PROCESS] OF I_Process_LinkedList;  // access to all linked lists for process entry
  _ListResult             : ST_PROCESS_LIST_RESULT;
  _ProcessData            : ST_PROCESS_DATA;

  {attribute 'displaymode':='bin'}
  _wTargetMask            : ARRAY[1..SIZEOF(T_PROCESS)*8] OF BYTE; // bits for PosStop[] to use in XtsStation of target process

  _stMsg                  : ST_Message;
  _MessageLevel           : E_MessageType;
END_VAR

METHOD Check : BOOL // call this method in the extending/inheriting class
VAR_INST
  _eCommandOld    : E_INSTANCE_CMD;
END_VAR
//-----------------------------------------------------------------------------
//-----------------------------------------------------------------------------
// plausibility checks
//-----------------------------------------------------------------------------
IF NOT (_nProcess > 0)
THEN
  _eCheck                 := E_INSTANCE_CHECK.INVALID_PROCESS_ID_ZERO;
  RETURN;
END_IF

IF NOT (_nProcess < E_INSTANCE.INSTANCE_MAX)
THEN
  _eCheck                 := E_INSTANCE_CHECK.INVALID_PROCESS_ID_MAX;
  RETURN;
END_IF
//-----------------------------------------------------------------------------
//-----------------------------------------------------------------------------
// pointer checks
//-----------------------------------------------------------------------------
IF NOT __ISVALIDREF(_InstanceCtrl)
THEN
  _eCheck                 := E_INSTANCE_CHECK.INVALID_INSTANCE_CONTROL_REFERENCE;
  RETURN;
END_IF

IF NOT __ISVALIDREF(_InstanceState)
THEN
  _eCheck                 := E_INSTANCE_CHECK.INVALID_INSTANCE_STATE_REFERENCE;
  RETURN;
END_IF

IF NOT (_ItfProcessCollector[_nProcess] <> 0) 
THEN
  _eCheck                 := E_INSTANCE_CHECK.INVALID_INTERFACE_POINTER;
  RETURN;
END_IF

IF NOT (_ItfProcessCollector[_nProcess].ProcessId > 0)
THEN
  _eCheck                 := E_INSTANCE_CHECK.INVALID_PROCESS_ID_ZERO;
  RETURN;
END_IF

IF NOT (_ItfProcessCollector[_nProcess].ProcessId < E_INSTANCE.INSTANCE_MAX)
THEN
  _eCheck                 := E_INSTANCE_CHECK.INVALID_PROCESS_ID_MAX;
  RETURN;
END_IF

IF NOT (_nProcess = _ItfProcessCollector[_nProcess].ProcessId)
THEN
  _eCheck                 := E_INSTANCE_CHECK.INVALID_PROCESS_ID_NOTEQUAL_COLLECTOR_ID;
  RETURN;
END_IF

IF NOT (_ItfProcessList[_nProcess] <> 0)
THEN
  _eCheck                 := E_INSTANCE_CHECK.INVALID_INDEX_IN_LIST;
  RETURN;
END_IF
//-----------------------------------------------------------------------------
//-----------------------------------------------------------------------------
// connect datafields to interface of ProcessCollector
//-----------------------------------------------------------------------------
_ItfProcessCollector[_nProcess].ProcessCtrl   REF= _Ctrl;
_ItfProcessCollector[_nProcess].ProcessState  REF= _State;

//-----------------------------------------------------------------------------
//-----------------------------------------------------------------------------
// set message device
//-----------------------------------------------------------------------------
_stMsg.eDevice            := e_Device.Process + TO_UINT(_nProcess);
//-----------------------------------------------------------------------------
//-----------------------------------------------------------------------------
// log cmd change
//-----------------------------------------------------------------------------
IF _eCmd <> _eCommandOld
THEN
  _eCommandOld              := _eCmd;

  IF (_MessageLevel = E_MessageType.eMessageVerbose)
  THEN
    _stMsg.eType            := E_MessageType.eMessageVerbose;
    _stMsg.eSubdevice       := e_Subdevice.Instance_Command;
    _stMsg.iErrorNumber     := _nProcess;
    _stMsg.sText            := concat(TO_STRING(_nProcess), ': ');
    _stMsg.sText            := concat(_stMsg.sText, TO_STRING(_eCmd));
    f_MessageSet(_stMsg);
  END_IF
END_IF
//-----------------------------------------------------------------------------
//-----------------------------------------------------------------------------
_eCheck                   := E_INSTANCE_CHECK.CHECK_DONE;
Check                     := TRUE;
END_METHOD

PROPERTY CollectorInterface : array[1..MAX_PROCESS] of I_ProcessCollector
SET
_ItfProcessCollector := CollectorInterface;
END_SET
END_PROPERTY

PROPERTY InstanceCtrl : REFERENCE TO ARRAY[1..MAX_PROCESS] OF ST_INSTANCE_CTRL
SET
_InstanceCtrl ref= InstanceCtrl;
END_SET
END_PROPERTY

PROPERTY InstanceState : REFERENCE TO ARRAY[1..MAX_PROCESS] OF ST_INSTANCE_STATE
SET
_InstanceState ref= InstanceState;
END_SET
END_PROPERTY

PROPERTY MessageLevel : e_MessageType
SET
VAR
  _mlidx      : UINT;
END_VAR
IF NOT Check() THEN RETURN; END_IF
//-----------------------------------------------------------------------------
//-----------------------------------------------------------------------------
// message levels for underlying ProcessCollector and XtsStations
//-----------------------------------------------------------------------------
//-----------------------------------------------------------------------------
_MessageLevel                                 :=  MessageLevel;
GVL_MSG.MessageLevelProcess[_nProcess]        := _MessageLevel;

FOR _mlidx := _ItfProcessCollector[_nProcess].StationFirst 
           TO _ItfProcessCollector[_nProcess].StationLast
DO
  GVL_MSG.MessageLevelStations[_mlidx]        := _MessageLevel;
END_FOR
END_SET
END_PROPERTY

PROPERTY ProcessId : E_INSTANCE
GET
ProcessId := _nProcess;
END_GET
SET
_nProcess := ProcessId;
END_SET
END_PROPERTY

PROPERTY ProcessLinkedLists : ARRAY[1..max_process] OF I_Process_LinkedList
SET
_ItfProcessList := ProcessLinkedLists;
END_SET
END_PROPERTY

END_FUNCTION_BLOCK

// ---- XTS/XtsTransportUnit/fb_TransportUnit.TcPOU
//---------------------------------------------------------------------------------------------------------------
//
//  HAUD 2024.03.18
//
//  - XTS_TRANSPORT_LAYER
//
//  fb_TransportUnit
//  - Ctrl/STate interface, reacts to change of command
//    - Cmd(E_TRANSPORT_CTRL)
//
//  - controls members via structures and interfaces for getting XTS in defined state
//    - CMD_INIT:
//        - XPU is initialized:         XTS_CMD_INIT + PROGRESS_DONE
//        - XPU cyclic checks enabled:  XTS_IDLE     + PROGRESS_WORKING
//        - XPU detects mover:          _XpuState.Check == MOVER_ID_DETECTION_VALID
//
//    - CMD_IDLE
//      - Cyclic Checks of XPU and CaGroup
//        - XPU cyclic checks enabled:  XTS_IDLE     + PROGRESS_WORKING
//
//
//  CTRL / STATE --> see proprerties
//  structs for use of function block via mapping
//  cyclic check for new command
//
//  VAR INPUT / OUTPUT --> see properties
//
//---------------------------------------------------------------------------------------------------------------
// This SOFTWARE is provided as an Exemple by THE PROVIDER "as is" and "with all faults." THE PROVIDER makes no 
// representations or warranties of any kind concerning the safety, suitability, lack of viruses, inaccuracies, 
// typographical errors, or other harmful components of this SOFTWARE. There are inherent dangers in the use of 
// any software, and you are solely responsible for determining whether this SOFTWARE is compatible with your 
// equipment and other software installed on your equipment. You are also solely responsible for the protection 
// of your equipment and backup of your data, and THE PROVIDER will not be liable for any damages you may suffer 
// in connection with using, modifying, or distributing this SOFTWARE.
//---------------------------------------------------------------------------------------------------------------
FUNCTION_BLOCK fb_TransportUnit
VAR
  _eCheck                       : E_XTS_TRANSPORT_CHECK;

  // Transport Ctrl/State
  _Ctrl                         : REFERENCE TO ST_XTS_TRANSPORT_CTRL;
  _State                        : REFERENCE TO ST_XTS_TRANSPORT_STATE;


  // execute transport commands
  _eCmd,
  _eCmdOld                      : E_XTS_TRANSPORT_CTRL;

  // execution state
  _eState                       : E_XTS_TRANSPORT_STATE;

  // execution result
  _eJobResult,
  _eResult                      : E_PROGRESS;


  // members of transport
  _XpuCtrl                      : REFERENCE TO ST_XPU_CTRL;                     // processing unit ctrl
  _XpuState                     : REFERENCE TO ST_XPU_STATE;                    // processing unit state
  _XpuInfo                      : REFERENCE TO ST_XPU_INFO;                     // processing unit information

  _GroupItf                     : I_XtsTransport_CaGroup;                       // group methods
  _GroupInfo                    : REFERENCE TO ST_GROUP_INFO;                   // info from group

  _MoverItf                     : REFERENCE TO ARRAY[1..MAX_MOVER] OF I_XtsTransport_Mover;   // mover methods
  _MoverInfo                    : REFERENCE TO ARRAY[1..MAX_MOVER] OF ST_MOVER_INFO;          // info from mover
  _MoverLastPosition            : REFERENCE TO ARRAY[1..MAX_MOVER] OF LREAL;                  // last commanded position of mover
  _MoverLastGap                 : REFERENCE TO ARRAY[1..MAX_MOVER] OF LREAL;                  // last commanded gapp of mover

  _StationStart                 : REFERENCE TO ST_STATION_PARAMETER;            // position, gap, dynamic constraints for sending all mover to start position

  // stations lists
  _ItfStationList               : REFERENCE TO ARRAY[1..MAX_STATION]  OF I_Station_LinkedList;  // access to all stations lists

  // station controls
  _StationControl               : REFERENCE TO ARRAY[1..MAX_STATION]  OF ST_STATION_CTRL;

  // station states
  _StationState                 : REFERENCE TO ARRAY[1..MAX_STATION]  OF ST_STATION_STATE;


  // access to stations methods by interface
  _ItfStationCtrl               : REFERENCE TO ARRAY[1..MAX_STATION]  OF I_XtsTransport_Station;

  _nStartStation                : UINT;

  _stMoverDataSend              : ST_STATION_MOVER_DATA;    // mover ticket data

  _stListResult                 : ST_STATION_LIST_RESULT;   // Xts station linkedlist entry

  _eMessageLevel                : E_MessageType;
  _stMsg                        : ST_Message;
END_VAR

IF NOT Check() THEN RETURN; END_IF

_stMsg.eDevice                  := XtsTransportUnit + 1;

_eCmd                           := _Ctrl.Cmd;
// check for command change
// get state for cmd
IF (_eCmd <> _eCmdOld)
THEN
  _eState                       := Cmd(_eCmd);
  _eCmdOld                      := _eCmd;

  IF (_eMessageLevel = E_MessageType.eMessageVerbose)
  THEN
    _stMsg.eType                := E_MessageType.eMessageVerbose;
    _stMsg.eSubdevice           := e_Subdevice.TransportUnit_General;
    _stMsg.iErrorNumber         := 0;
    _stMsg.sText                := concat( 'Command: ', TO_STRING(_eCmd));
    _stMsg.sText                := concat(_stMsg.sText, ': ');
    _stMsg.sText                := concat(_stMsg.sText, TO_STRING(_eResult));
    f_MessageSet(_stMsg);
  END_IF
END_IF

CASE _eResult
OF
  E_PROGRESS.PROGRESS_INVALID:
    _State.State                := TO_UINT(_eResult);

  E_PROGRESS.PROGRESS_ERROR:
    _State.State                := _eState + E_PROGRESS.PROGRESS_ERROR;

  E_PROGRESS.PROGRESS_DONE:
    _State.State                := _eState + E_PROGRESS.PROGRESS_DONE;

    IF (_GroupInfo.GroupErrorStop) OR
       (_GroupInfo.GroupError)     OR
       NOT (_XpuInfo.AllPositionsValid)
    THEN
      _eResult                  := E_PROGRESS.PROGRESS_ERROR;
    END_IF
ELSE
  _State.State                  := _eState + _eResult;

  CASE _eState
  OF
    E_XTS_TRANSPORT_STATE.TRANSPORT_INIT:
      _eResult                  := XpuInit(TRUE);
  
    E_XTS_TRANSPORT_STATE.TRANSPORT_IDLE:
      _eResult                  := f_GetProgress(_XpuState.State);
  
      IF (_GroupInfo.GroupErrorStop) OR
         (_GroupInfo.GroupError)     OR
         NOT (_XpuInfo.AllPositionsValid)
      THEN
        _eResult                := E_PROGRESS.PROGRESS_ERROR;
      END_IF
  
    E_XTS_TRANSPORT_STATE.TRANSPORT_MOVER_ENABLE:
      IF NOT (_XpuState.DcLink)
      THEN
        _eResult                := E_PROGRESS.PROGRESS_BUSY;

      ELSIF NOT (_XpuInfo.AllPositionsValid)
      THEN
        _eResult                := E_PROGRESS.PROGRESS_ERROR;
      ELSE
        _eResult                := MoverEnableAll(TRUE);
      END_IF
  
    E_XTS_TRANSPORT_STATE.TRANSPORT_MOVER_DISABLE:
      _eResult                  := MoverDisableAll(TRUE);

    E_XTS_TRANSPORT_STATE.TRANSPORT_MOVER_HALT_CA:
      _eResult                  := MoverHaltAll(TRUE);

    E_XTS_TRANSPORT_STATE.TRANSPORT_MOVER_STOP:
      _eResult                  := MoverStopAll(TRUE);
  
    E_XTS_TRANSPORT_STATE.TRANSPORT_GROUP_CLEAR:
      _eResult                  := GroupClear(TRUE);
  
    E_XTS_TRANSPORT_STATE.TRANSPORT_GROUP_BUILD:
      _eResult                  := GroupBuild(TRUE);
  
    E_XTS_TRANSPORT_STATE.TRANSPORT_GROUP_ENABLE:
      _eResult                  := GroupEnable(TRUE);

    E_XTS_TRANSPORT_STATE.TRANSPORT_GROUP_STOP:
      _eResult                  := GroupStop(TRUE);

    E_XTS_TRANSPORT_STATE.TRANSPORT_START:
      IF NOT (_XpuState.DcLink)
      THEN
        _eResult                := E_PROGRESS.PROGRESS_BUSY;

      ELSIF NOT (_XpuInfo.AllPositionsValid)
      THEN
        _eResult                := E_PROGRESS.PROGRESS_ERROR;
      ELSE
        _eResult                := TransportStart(TRUE);
      END_IF
  
    E_XTS_TRANSPORT_STATE.TRANSPORT_RESTART:
      IF NOT (_XpuState.DcLink)
      THEN
        _eResult                := E_PROGRESS.PROGRESS_BUSY;

      ELSIF NOT (_XpuInfo.AllPositionsValid)
      THEN
        _eResult                := E_PROGRESS.PROGRESS_ERROR;
      ELSE
        _eResult                := TransportRestart(TRUE);
      END_IF
  ELSE
    _eResult                    := E_PROGRESS.PROGRESS_INVALID;
  END_CASE

END_CASE

_State.XpuState                 := _XpuState;
_State.XpuInfo                  := _XpuInfo;
_State.GroupInfo                := _GroupInfo;

METHOD PRIVATE Check  : BOOL
VAR_INST
  _idx        : UINT;
END_VAR

IF NOT __ISVALIDREF(_Ctrl)
THEN
  _eCheck                     := E_XTS_TRANSPORT_CHECK.POINTER_NULL_CTRL;
  RETURN;
END_IF

IF NOT __ISVALIDREF(_State)
THEN
  _eCheck                     := E_XTS_TRANSPORT_CHECK.POINTER_NULL_STATE;
  RETURN;
END_IF

_State.Check                  := _eCheck;

IF NOT __ISVALIDREF(_XpuCtrl)
THEN
  _eCheck                     := E_XTS_TRANSPORT_CHECK.POINTER_NULL_XPU_CTRL;
  RETURN;
END_IF

IF NOT __ISVALIDREF(_XpuState)
THEN
  _eCheck                     := E_XTS_TRANSPORT_CHECK.POINTER_NULL_XPU_STATE;
  RETURN;
END_IF

IF NOT __ISVALIDREF(_XpuInfo)
THEN
  _eCheck                     := E_XTS_TRANSPORT_CHECK.POINTER_NULL_XPU_INFO;
  RETURN;
END_IF

IF NOT (_GroupItf <> 0)
THEN
  _eCheck                     := E_XTS_TRANSPORT_CHECK.POINTER_NULL_GROUP_ITF;
  RETURN;
END_IF

IF NOT __ISVALIDREF(_GroupInfo)
THEN
  _eCheck                     := E_XTS_TRANSPORT_CHECK.POINTER_NULL_GROUP_INFO;
  RETURN;
END_IF

IF NOT __ISVALIDREF(_MoverItf)
THEN
  _eCheck                     := E_XTS_TRANSPORT_CHECK.POINTER_NULL_MOVER;
  RETURN;
END_IF

FOR _idx := 1 TO MAX_MOVER
DO
  IF NOT (_MoverItf[_idx] <> 0)
  THEN
    _eCheck                   := E_XTS_TRANSPORT_CHECK.POINTER_NULL_MOVER_ITF;
    RETURN;
  END_IF
END_FOR

IF NOT __ISVALIDREF(_MoverInfo)
THEN
  _eCheck                     := E_XTS_TRANSPORT_CHECK.POINTER_NULL_MOVER_INFO;
  RETURN;
END_IF

IF NOT __ISVALIDREF(_MoverLastPosition)
THEN
  _eCheck                     := E_XTS_TRANSPORT_CHECK.POINTER_NULL_MOVER_LAST_POS;
  RETURN;
END_IF

IF NOT __ISVALIDREF(_MoverLastGap)
THEN
  _eCheck                     := E_XTS_TRANSPORT_CHECK.POINTER_NULL_MOVER_LAST_GAP;
  RETURN;
END_IF

IF NOT __ISVALIDREF(_StationStart)
THEN
  _eCheck                     := E_XTS_TRANSPORT_CHECK.POINTER_NULL_STATION_START;
  RETURN;
END_IF

IF NOT __ISVALIDREF(_ItfStationList)
THEN
  _eCheck                     := E_XTS_TRANSPORT_CHECK.POINTER_NULL_STATION_ITF;
  RETURN;
END_IF

IF NOT __ISVALIDREF(_StationControl)
THEN
  _eCheck                     := E_XTS_TRANSPORT_CHECK.POINTER_NULL_STATION_CONTROL;
  RETURN;
END_IF

IF NOT __ISVALIDREF(_StationState)
THEN
  _eCheck                     := E_XTS_TRANSPORT_CHECK.POINTER_NULL_STATION_STATE;
  RETURN;
END_IF

IF NOT __ISVALIDREF(_ItfStationCtrl)
THEN
  _eCheck                     := E_XTS_TRANSPORT_CHECK.POINTER_NULL_STATION_CTRL_ITF;
  RETURN;
END_IF


_eCheck                       := E_XTS_TRANSPORT_CHECK.DONE_CHECK;
Check                         := TRUE;
END_METHOD

METHOD PRIVATE Cmd : E_XTS_TRANSPORT_STATE
VAR_INPUT
  Ctrl      : E_XTS_TRANSPORT_CTRL;
END_VAR
VAR_INST
  _eState   : E_XTS_TRANSPORT_STATE;
END_VAR
IF NOT Check() THEN RETURN; END_IF


CASE Ctrl
OF
  E_XTS_TRANSPORT_CTRL.CMD_NULL:  // clear all method calls
    _eState               := E_XTS_TRANSPORT_STATE.TRANSPORT_NULL;
    _eResult              := XpuInit         (FALSE);
    _eResult              := GroupClear      (FALSE);
    _eResult              := GroupBuild      (FALSE);
    _eResult              := GroupEnable     (FALSE);
    _eResult              := GroupStop       (FALSE);
    _eResult              := MoverEnableAll  (FALSE);
    _eResult              := MoverDisableAll (FALSE);
    _eResult              := MoverHaltAll    (FALSE);
    _eResult              := MoverStopAll    (FALSE);
    _eResult              := TransportStart  (FALSE);
    _eResult              := TransportRestart(FALSE);

  E_XTS_TRANSPORT_CTRL.CMD_INIT:  // clear methods for initialization
    _eState               := E_XTS_TRANSPORT_STATE.TRANSPORT_INIT;
    _eResult              := XpuInit(FALSE);


ELSE
  IF NOT (_XpuState.Init = E_XPU_INIT.INIT_DONE)
  THEN
    // no init, no further commands possible
    _eState               := E_XTS_TRANSPORT_STATE.TRANSPORT_INVALID;
  ELSE
    CASE Ctrl
    OF
      E_XTS_TRANSPORT_CTRL.CMD_IDLE:
        _eState           := E_XTS_TRANSPORT_STATE.TRANSPORT_IDLE;

      E_XTS_TRANSPORT_CTRL.CMD_MOVER_ENABLE:
        _eState           := E_XTS_TRANSPORT_STATE.TRANSPORT_MOVER_ENABLE;
        _eResult          := MoverEnableAll(FALSE);

      E_XTS_TRANSPORT_CTRL.CMD_MOVER_DISABLE:
        _eState           := E_XTS_TRANSPORT_STATE.TRANSPORT_MOVER_DISABLE;
        _eResult          := MoverDisableAll(FALSE);

      E_XTS_TRANSPORT_CTRL.CMD_MOVER_HALT_CA:
        _eState           := E_XTS_TRANSPORT_STATE.TRANSPORT_MOVER_HALT_CA;
        _eResult          := MoverHaltAll(FALSE);

      E_XTS_TRANSPORT_CTRL.CMD_MOVER_STOP:
        _eState           := E_XTS_TRANSPORT_STATE.TRANSPORT_MOVER_STOP;
        _eResult          := MoverStopAll(FALSE);

      E_XTS_TRANSPORT_CTRL.CMD_GROUP_CLEAR:
        _eState           := E_XTS_TRANSPORT_STATE.TRANSPORT_GROUP_CLEAR;
        _eResult          := GroupClear (FALSE);

      E_XTS_TRANSPORT_CTRL.CMD_GROUP_BUILD:
        _eState           := E_XTS_TRANSPORT_STATE.TRANSPORT_GROUP_BUILD;
        _eResult          := GroupBuild (FALSE);

      E_XTS_TRANSPORT_CTRL.CMD_GROUP_ENABLE:
        _eState           := E_XTS_TRANSPORT_STATE.TRANSPORT_GROUP_ENABLE;
        _eResult          := GroupEnable(FALSE);

      E_XTS_TRANSPORT_CTRL.CMD_GROUP_STOP:
        _eState           := E_XTS_TRANSPORT_STATE.TRANSPORT_GROUP_STOP;
        _eResult          := GroupStop(FALSE);

      E_XTS_TRANSPORT_CTRL.CMD_TRANSPORT_START:
        _eState           := E_XTS_TRANSPORT_STATE.TRANSPORT_START;
        _eResult          := TransportStart(FALSE);

      E_XTS_TRANSPORT_CTRL.CMD_TRANSPORT_RESTART:
        _eState           := E_XTS_TRANSPORT_STATE.TRANSPORT_RESTART;
        _eResult          := TransportRestart(FALSE);

    ELSE
        _eState           := E_XTS_TRANSPORT_STATE.TRANSPORT_INVALID;
    END_CASE
  END_IF
END_CASE

Cmd                       := _eState;
END_METHOD

PROPERTY Ctrl : REFERENCE TO ST_XTS_TRANSPORT_CTRL
SET
_Ctrl REF= Ctrl;
END_SET
END_PROPERTY

METHOD GroupBuild : E_PROGRESS
VAR_INPUT
  Execute     : BOOL;
END_VAR
VAR_INST
  _nErrorId   : UDINT;
  _eJobReslt,
  _eState     : E_PROGRESS;
END_VAR
//-----------------------------------------------------------------------------
IF NOT Execute 
THEN 
	_eState                       := E_PROGRESS.PROGRESS_INIT; 
END_IF 
//-----------------------------------------------------------------------------
IF NOT Check() 
THEN 
	GroupBuild                    := E_PROGRESS.PROGRESS_ERROR; 
	RETURN; 
END_IF
//-----------------------------------------------------------------------------
//-----------------------------------------------------------------------------
CASE _eState
OF
  E_PROGRESS.PROGRESS_INIT:
    IF Execute
    THEN
      _nErrorId                 := 0;

      IF (_GroupInfo.AxisCount <> 0)
      THEN
        _nErrorId               := 9999;
        _eState                 := E_PROGRESS.PROGRESS_ERROR;
      ELSE
        _eState                 := E_PROGRESS.PROGRESS_BUSY;
        _eJobReslt              := _GroupItf.AddAll(FALSE);
      END_IF
    END_IF
END_CASE
//---------------------------------------------------------------------------
//---------------------------------------------------------------------------
CASE _eState
OF
  E_PROGRESS.PROGRESS_BUSY:
    _eJobReslt                  := _GroupItf.AddAll(TRUE);

    IF (_eJobReslt = E_PROGRESS.PROGRESS_ERROR)
    THEN
      _eState                   := E_PROGRESS.PROGRESS_ERROR;

      _nErrorId                 := _GroupInfo.GroupErrorId;
      _eJobReslt                := _GroupItf.AddAll(FALSE);

    ELSIF (_eJobReslt = E_PROGRESS.PROGRESS_DONE)
    THEN
      _eState                   := E_PROGRESS.PROGRESS_PREPARE;
      _eJobReslt                := _GroupItf.AddAll(FALSE);
	  _eJobReslt				:= _GroupItf.Reset(FALSE);
    END_IF
END_CASE
//-----------------------------------------------------------------------------
//-----------------------------------------------------------------------------
CASE _eState
OF
  E_PROGRESS.PROGRESS_PREPARE:
    _eJobReslt                  := _GroupItf.Reset(TRUE);

    IF (_eJobReslt = E_PROGRESS.PROGRESS_ERROR)
    THEN
      _eState                   := E_PROGRESS.PROGRESS_ERROR;

      _nErrorId                 := _GroupInfo.GroupErrorId;
	    _eJobReslt				        := _GroupItf.Reset(FALSE);

    ELSIF (_eJobReslt = E_PROGRESS.PROGRESS_DONE)
    THEN
      _eState                   := E_PROGRESS.PROGRESS_DONE;
	    _eJobReslt				        := _GroupItf.Reset(FALSE);

      IF (_eMessageLevel = E_MessageType.eMessageVerbose)
      THEN
        _stMsg.eType            := E_MessageType.eMessageVerbose;
        _stMsg.eSubdevice       := e_Subdevice.TransportUnit_General;
        _stMsg.iErrorNumber     := 0;
        _stMsg.sText            := concat( 'State: ', TO_STRING(THIS^._eState));
        _stMsg.sText            := concat(_stMsg.sText, ': ');
        _stMsg.sText            := concat(_stMsg.sText, TO_STRING(_eState));
        f_MessageSet(_stMsg);
      END_IF
    END_IF
END_CASE
//-----------------------------------------------------------------------------
//-----------------------------------------------------------------------------

GroupBuild                      := _eState;
END_METHOD

METHOD GroupClear : E_PROGRESS
VAR_INPUT
  Execute     : BOOL;
END_VAR
VAR_INST
  _nRepeat,
  _nStation,
  _nErrorId   : UDINT;
  _eJobReslt,
  _eState     : E_PROGRESS;
END_VAR
//-----------------------------------------------------------------------------
IF NOT Execute 
THEN 
	_eState                       := E_PROGRESS.PROGRESS_INIT; 
END_IF 
//-----------------------------------------------------------------------------
IF NOT Check() 
THEN 
	GroupClear                    := E_PROGRESS.PROGRESS_ERROR; 
	RETURN; 
END_IF
//-----------------------------------------------------------------------------
//-----------------------------------------------------------------------------
CASE _eState
OF
  E_PROGRESS.PROGRESS_INIT:
    IF Execute
    THEN
      _nRepeat                  :=
      _nErrorId                 := 0;
      _eJobReslt                := _GroupItf.McHaltAll(FALSE);
      _eJobReslt                := _GroupItf.RemoveAll(FALSE);
      _eJobReslt                := _GroupItf.McResetAll(FALSE);
      _eJobReslt                := _GroupItf.Disable(FALSE);
      _eJobReslt                := _GroupItf.Reset(FALSE);

      _eState                   := E_PROGRESS.PROGRESS_BUSY;
    END_IF
END_CASE
//---------------------------------------------------------------------------
//---------------------------------------------------------------------------
CASE _eState
OF
  E_PROGRESS.PROGRESS_BUSY:
    _eJobReslt                  := _GroupItf.McHaltAll(TRUE);

    IF (_eJobReslt = E_PROGRESS.PROGRESS_ERROR)
    THEN
      _eState                   := E_PROGRESS.PROGRESS_STARTUP;
      _nErrorId                 := _GroupInfo.GroupErrorId;
      _eJobReslt                := _GroupItf.McHaltAll(FALSE);

    ELSIF (_eJobReslt = E_PROGRESS.PROGRESS_DONE)
    THEN
      _eState                   := E_PROGRESS.PROGRESS_STARTUP;
      _eJobReslt                := _GroupItf.McHaltAll(FALSE);
    END_IF
  //---------------------------------------------------------------------------
  //---------------------------------------------------------------------------
  E_PROGRESS.PROGRESS_PREPARE:
    _eJobReslt                  := _GroupItf.McResetAll(TRUE);

    IF (_eJobReslt = E_PROGRESS.PROGRESS_DONE)
    THEN
      _eState                   := E_PROGRESS.PROGRESS_CHECK;
      _eJobReslt                := _GroupItf.McResetAll(FALSE);
    END_IF
  //---------------------------------------------------------------------------
  //---------------------------------------------------------------------------
  E_PROGRESS.PROGRESS_STARTUP:
    _eJobReslt                  := _GroupItf.RemoveAll(TRUE);

    IF (_eJobReslt = E_PROGRESS.PROGRESS_ERROR)
    THEN
      _eState                   := E_PROGRESS.PROGRESS_ERROR;
      _nErrorId                 := _GroupInfo.GroupErrorId;
      _eJobReslt                := _GroupItf.RemoveAll(FALSE);

    ELSIF (_eJobReslt = E_PROGRESS.PROGRESS_DONE)
    THEN
      _eState                   := E_PROGRESS.PROGRESS_PREPARE;
      _eJobReslt                := _GroupItf.RemoveAll(FALSE);
    END_IF
  //---------------------------------------------------------------------------
  //---------------------------------------------------------------------------
  E_PROGRESS.PROGRESS_CHECK:
    _eJobReslt                  := _GroupItf.Disable(TRUE);

    IF (_eJobReslt = E_PROGRESS.PROGRESS_ERROR)
    THEN
      _eState                   := E_PROGRESS.PROGRESS_ERROR;
      _nErrorId                 := _GroupInfo.GroupErrorId;
      _eJobReslt                := _GroupItf.Disable(FALSE);

    ELSIF (_eJobReslt = E_PROGRESS.PROGRESS_DONE)
    THEN
      _eState                   := E_PROGRESS.PROGRESS_OCCUPIED;
      _eJobReslt                := _GroupItf.Disable(FALSE);
    END_IF
  //---------------------------------------------------------------------------
  //---------------------------------------------------------------------------
  E_PROGRESS.PROGRESS_OCCUPIED:
    _eJobReslt                  := _GroupItf.Reset(TRUE);

    IF (_eJobReslt = E_PROGRESS.PROGRESS_ERROR)
    THEN
      _eState                   := E_PROGRESS.PROGRESS_ERROR;
      _nErrorId                 := _GroupInfo.GroupErrorId;
      _eJobReslt                := _GroupItf.Reset(FALSE);

    ELSIF (_eJobReslt = E_PROGRESS.PROGRESS_DONE)
    THEN
      _eState                   := E_PROGRESS.PROGRESS_WORKING;
      _eJobReslt                := _GroupItf.Reset(FALSE);
    END_IF
END_CASE
//-----------------------------------------------------------------------------
//-----------------------------------------------------------------------------
CASE _eState
OF
  E_PROGRESS.PROGRESS_WORKING:
    IF (_GroupInfo.CaGroupState = E_CA_GROUP_STATE.mcGroupStateDisabled) AND NOT
       (_GroupInfo.GroupError)
    THEN
      _eState                   := E_PROGRESS.PROGRESS_DONE;

      IF (_eMessageLevel = E_MessageType.eMessageVerbose)
      THEN
        _stMsg.eType            := E_MessageType.eMessageVerbose;
        _stMsg.eSubdevice       := e_Subdevice.TransportUnit_General;
        _stMsg.iErrorNumber     := 0;
        _stMsg.sText            := concat( 'State: ', TO_STRING(THIS^._eState));
        _stMsg.sText            := concat(_stMsg.sText, ': ');
        _stMsg.sText            := concat(_stMsg.sText, TO_STRING(_eState));
        f_MessageSet(_stMsg);
      END_IF
    ELSE
      _nRepeat                  := _nRepeat + 1;
      IF NOT (_nRepeat > 2)
      THEN
        _eState                 := E_PROGRESS.PROGRESS_PREPARE;
      ELSE
        _eState                 := E_PROGRESS.PROGRESS_ERROR;
      END_IF
    END_IF
END_CASE
//-----------------------------------------------------------------------------
//-----------------------------------------------------------------------------

GroupClear                      := _eState;
END_METHOD

METHOD GroupEnable : E_PROGRESS
VAR_INPUT
  Execute     : BOOL;
END_VAR
VAR_INST
  _nErrorId   : UDINT;
  _eJobReslt,
  _eState     : E_PROGRESS;
END_VAR
//-----------------------------------------------------------------------------
IF NOT Execute 
THEN 
	_eState                       := E_PROGRESS.PROGRESS_INIT; 
END_IF 
//-----------------------------------------------------------------------------
IF NOT Check() 
THEN 
	GroupEnable                   := E_PROGRESS.PROGRESS_ERROR; 
	RETURN; 
END_IF
//-----------------------------------------------------------------------------
//-----------------------------------------------------------------------------
CASE _eState
OF
  E_PROGRESS.PROGRESS_INIT:
    IF Execute
    THEN
      _nErrorId                 := 0;

      IF NOT (_GroupInfo.AxisCount <> 0)
      THEN
        _nErrorId               := 9999;
        _eState                 := E_PROGRESS.PROGRESS_ERROR;
      ELSE
        _eState                 := E_PROGRESS.PROGRESS_BUSY;
        _eJobReslt              := _GroupItf.Enable(FALSE);
      END_IF
    END_IF
END_CASE
//---------------------------------------------------------------------------
//---------------------------------------------------------------------------
CASE _eState
OF
  E_PROGRESS.PROGRESS_BUSY:
    _eJobReslt                  := _GroupItf.Enable(TRUE);

    IF (_eJobReslt = E_PROGRESS.PROGRESS_ERROR)
    THEN
      _eState                   := E_PROGRESS.PROGRESS_ERROR;

      _nErrorId                 := _GroupInfo.GroupErrorId;
      _eJobReslt                := _GroupItf.Enable(FALSE);

    ELSIF (_eJobReslt = E_PROGRESS.PROGRESS_DONE)
    THEN
      _eState                   := E_PROGRESS.PROGRESS_CHECK;
      _eJobReslt                := _GroupItf.Enable(FALSE);
    END_IF
END_CASE
//-----------------------------------------------------------------------------
//-----------------------------------------------------------------------------
CASE _eState
OF
  E_PROGRESS.PROGRESS_CHECK:
    IF (_GroupInfo.GroupStandby) OR
       (_GroupInfo.GroupMoving)  OR
       (_GroupInfo.GroupNotReady)
    THEN
      _eState                   := E_PROGRESS.PROGRESS_DONE;

      IF (_eMessageLevel = E_MessageType.eMessageVerbose)
      THEN
        _stMsg.eType            := E_MessageType.eMessageVerbose;
        _stMsg.eSubdevice       := e_Subdevice.TransportUnit_General;
        _stMsg.iErrorNumber     := 0;
        _stMsg.sText            := concat( 'State: ', TO_STRING(THIS^._eState));
        _stMsg.sText            := concat(_stMsg.sText, ': ');
        _stMsg.sText            := concat(_stMsg.sText, TO_STRING(_eState));
        f_MessageSet(_stMsg);
      END_IF
    ELSE
      IF (_GroupInfo.GroupErrorStop) OR
         (_GroupInfo.GroupError)
      THEN
        _eState                 := E_PROGRESS.PROGRESS_ERROR;
      END_IF
    END_IF
END_CASE
//-----------------------------------------------------------------------------
//-----------------------------------------------------------------------------
GroupEnable                     := _eState;
END_METHOD

PROPERTY GroupInfo : REFERENCE TO ST_GROUP_INFO
SET
_GroupInfo REF= GroupInfo;
END_SET
END_PROPERTY

PROPERTY GroupItf : I_XtsTransport_CaGroup
SET
_GroupItf := GroupItf;
END_SET
END_PROPERTY

METHOD GroupStop : E_PROGRESS
VAR_INPUT
  Execute     : BOOL;
END_VAR
VAR_INST
  _nRepeat,
  _nStation,
  _nErrorId   : UDINT;
  _eJobReslt,
  _eState     : E_PROGRESS;
END_VAR
//-----------------------------------------------------------------------------
IF NOT Execute 
THEN 
	_eState                      := E_PROGRESS.PROGRESS_INIT; 
END_IF 
//-----------------------------------------------------------------------------
IF NOT Check() 
THEN 
	GroupStop                    := E_PROGRESS.PROGRESS_ERROR; 
	RETURN; 
END_IF
//-----------------------------------------------------------------------------
//-----------------------------------------------------------------------------
CASE _eState
OF
  E_PROGRESS.PROGRESS_INIT:
    IF Execute
    THEN
      _nRepeat                  :=
      _nErrorId                 := 0;
      _eJobReslt                := _GroupItf.Stop(FALSE);

      _eState                   := E_PROGRESS.PROGRESS_BUSY;
    END_IF
END_CASE
//---------------------------------------------------------------------------
//---------------------------------------------------------------------------
CASE _eState
OF
  E_PROGRESS.PROGRESS_BUSY:
    _eJobReslt                  := _GroupItf.Stop(TRUE);

    IF (_eJobReslt = E_PROGRESS.PROGRESS_ERROR)
    THEN
      _eState                   := E_PROGRESS.PROGRESS_PREPARE;
      _nErrorId                 := _GroupInfo.GroupErrorId;
      _eJobReslt                := _GroupItf.Stop(FALSE);

    ELSIF (_eJobReslt = E_PROGRESS.PROGRESS_DONE)
    THEN
      _eState                   := E_PROGRESS.PROGRESS_WORKING;
      _eJobReslt                := _GroupItf.Stop(FALSE);
    END_IF
END_CASE
//-----------------------------------------------------------------------------
//-----------------------------------------------------------------------------
CASE _eState
OF
  E_PROGRESS.PROGRESS_WORKING:
    IF NOT (_GroupInfo.GroupError)
    THEN
      _eState                   := E_PROGRESS.PROGRESS_DONE;

      IF (_eMessageLevel = E_MessageType.eMessageVerbose)
      THEN
        _stMsg.eType            := E_MessageType.eMessageVerbose;
        _stMsg.eSubdevice       := e_Subdevice.TransportUnit_General;
        _stMsg.iErrorNumber     := 0;
        _stMsg.sText            := concat( 'State: ', TO_STRING(THIS^._eState));
        _stMsg.sText            := concat(_stMsg.sText, ': ');
        _stMsg.sText            := concat(_stMsg.sText, TO_STRING(_eState));
        f_MessageSet(_stMsg);
      END_IF
    ELSE
      IF (_GroupInfo.GroupErrorStop) OR
         (_GroupInfo.GroupError)
      THEN
        _nRepeat                := _nRepeat + 1;
        IF NOT (_nRepeat > 2)
        THEN
          _eState               := E_PROGRESS.PROGRESS_BUSY;
        ELSE
          _eState               := E_PROGRESS.PROGRESS_ERROR;
        END_IF
      END_IF
    END_IF
END_CASE
//-----------------------------------------------------------------------------
//-----------------------------------------------------------------------------

GroupStop                       := _eState;
END_METHOD

PROPERTY MessageLevel : e_messagetype
SET
_eMessageLevel := MessageLevel;
END_SET
END_PROPERTY

METHOD MoverDisableAll : e_progress
VAR_INPUT
  Execute     : BOOL;
END_VAR
VAR_INST
  _nMover     : UINT;
  _nErrorId   : UDINT;
  _eRslt,
  _eState     : E_PROGRESS;
END_VAR
//-----------------------------------------------------------------------------
IF NOT Execute 
THEN 
	_eState                       := E_PROGRESS.PROGRESS_INIT; 
END_IF 
//-----------------------------------------------------------------------------
IF NOT Check() 
THEN 
	MoverDisableAll               := E_PROGRESS.PROGRESS_ERROR; 
	RETURN; 
END_IF
//-----------------------------------------------------------------------------
//-----------------------------------------------------------------------------
CASE _eState
OF
  E_PROGRESS.PROGRESS_INIT:
    IF Execute
    THEN
      _nErrorId                 := 0;
      _nMover                   := 1;

      _eState                   := E_PROGRESS.PROGRESS_BUSY;
    END_IF
END_CASE
//-----------------------------------------------------------------------------
//-----------------------------------------------------------------------------
CASE _eState
OF
  E_PROGRESS.PROGRESS_BUSY:
    _eState                     := E_PROGRESS.PROGRESS_PREPARE;
    _eRslt                      := _MoverItf[_nMover].Disable(FALSE);
END_CASE
//-----------------------------------------------------------------------------
//-----------------------------------------------------------------------------
CASE _eState
OF
  E_PROGRESS.PROGRESS_PREPARE:
    _eRslt                      := _MoverItf[_nMover].Disable(TRUE);

    IF (_eRslt = E_PROGRESS.PROGRESS_ERROR)
    THEN
      _eState                   := E_PROGRESS.PROGRESS_OCCUPIED;
      _nErrorId                 := _MoverInfo[_nMover].nErrorId; 
      _eRslt                    := _MoverItf[_nMover].Disable(FALSE);

    ELSIF (_eRslt = E_PROGRESS.PROGRESS_DONE)
    THEN
      _eState                   := E_PROGRESS.PROGRESS_STARTUP;
    END_IF
END_CASE
//-----------------------------------------------------------------------------
//-----------------------------------------------------------------------------
CASE _eState
OF
  E_PROGRESS.PROGRESS_STARTUP:
    _eState                     := E_PROGRESS.PROGRESS_CHECK;
    _eRslt                      := _MoverItf[_nMover].Disable(FALSE);


  E_PROGRESS.PROGRESS_OCCUPIED:
    _eRslt                      := _GroupItf.McResetAll(TRUE);

    IF (_eRslt = E_PROGRESS.PROGRESS_DONE)
    THEN
      _eState                   := E_PROGRESS.PROGRESS_PREPARE;
      _eRslt                    := _GroupItf.McResetAll(FALSE);
    END_IF
END_CASE
//-----------------------------------------------------------------------------
//-----------------------------------------------------------------------------
CASE _eState
OF
  E_PROGRESS.PROGRESS_CHECK:
    IF (_nMover > MAX_MOVER-1)
    THEN
      _eState                   := E_PROGRESS.PROGRESS_DONE;

      IF (_eMessageLevel = E_MessageType.eMessageVerbose)
      THEN
        _stMsg.eType            := E_MessageType.eMessageVerbose;
        _stMsg.eSubdevice       := e_Subdevice.TransportUnit_General;
        _stMsg.iErrorNumber     := 0;
        _stMsg.sText            := concat( 'State: ', TO_STRING(THIS^._eState));
        _stMsg.sText            := concat(_stMsg.sText, ': ');
        _stMsg.sText            := concat(_stMsg.sText, TO_STRING(_eState));
        f_MessageSet(_stMsg);
      END_IF
    ELSE
      _nMover                   := _nMover + 1;
      _eState                   := E_PROGRESS.PROGRESS_BUSY;
    END_IF
END_CASE
//-----------------------------------------------------------------------------
//-----------------------------------------------------------------------------

MoverDisableAll                 := _eState;
END_METHOD

METHOD MoverEnableAll : e_progress
VAR_INPUT
  Execute     : BOOL;
END_VAR
VAR_INST
  _nMover     : UINT;
  _nErrorId   : UDINT;
  _eRslt,
  _eState     : E_PROGRESS;
END_VAR
//-----------------------------------------------------------------------------
IF NOT Execute 
THEN 
	_eState                       := E_PROGRESS.PROGRESS_INIT; 
END_IF 
//-----------------------------------------------------------------------------
IF NOT Check() 
THEN 
	MoverEnableAll                := E_PROGRESS.PROGRESS_ERROR; 
	RETURN; 
END_IF
//-----------------------------------------------------------------------------
//-----------------------------------------------------------------------------
CASE _eState
OF
  E_PROGRESS.PROGRESS_INIT:
    IF Execute
    THEN
      _nErrorId                 := 0;
      _nMover                   := 1;

      _eState                   := E_PROGRESS.PROGRESS_BUSY;
    END_IF
END_CASE
//-----------------------------------------------------------------------------
//-----------------------------------------------------------------------------
CASE _eState
OF
  E_PROGRESS.PROGRESS_BUSY:
    _eState                     := E_PROGRESS.PROGRESS_PREPARE;
    _eRslt                      := _MoverItf[_nMover].Enable(FALSE);
END_CASE
//-----------------------------------------------------------------------------
//-----------------------------------------------------------------------------
CASE _eState
OF
  E_PROGRESS.PROGRESS_PREPARE:
    _eRslt                      := _MoverItf[_nMover].Enable(TRUE);

    IF (_eRslt = E_PROGRESS.PROGRESS_ERROR)
    THEN
      _eState                   := E_PROGRESS.PROGRESS_ERROR;
      _nErrorId                 := _MoverInfo[_nMover].nErrorId; 

    ELSIF (_eRslt = E_PROGRESS.PROGRESS_DONE)
    THEN
      _eState                   := E_PROGRESS.PROGRESS_STARTUP;
    END_IF
END_CASE
//-----------------------------------------------------------------------------
//-----------------------------------------------------------------------------
CASE _eState
OF
  E_PROGRESS.PROGRESS_STARTUP:
    _eState                     := E_PROGRESS.PROGRESS_CHECK;
    _eRslt                      := _MoverItf[_nMover].Enable(FALSE);
END_CASE
//-----------------------------------------------------------------------------
//-----------------------------------------------------------------------------
CASE _eState
OF
  E_PROGRESS.PROGRESS_CHECK:
    IF (_nMover > MAX_MOVER-1)
    THEN
      _eState                   := E_PROGRESS.PROGRESS_DONE;
      IF (_eMessageLevel = E_MessageType.eMessageVerbose)
      THEN
        _stMsg.eType            := E_MessageType.eMessageVerbose;
        _stMsg.eSubdevice       := e_Subdevice.TransportUnit_General;
        _stMsg.iErrorNumber     := 0;
        _stMsg.sText            := concat( 'State: ', TO_STRING(THIS^._eState));
        _stMsg.sText            := concat(_stMsg.sText, ': ');
        _stMsg.sText            := concat(_stMsg.sText, TO_STRING(_eState));
        f_MessageSet(_stMsg);
      END_IF
    ELSE
      _nMover                   := _nMover + 1;
      _eState                   := E_PROGRESS.PROGRESS_BUSY;
    END_IF
END_CASE
//-----------------------------------------------------------------------------
//-----------------------------------------------------------------------------

MoverEnableAll                  := _eState;
END_METHOD

METHOD MoverHaltAll : e_progress
VAR_INPUT
  Execute     : BOOL;
END_VAR
VAR_INST
  _nMover     : UINT;
  _nErrorId   : UDINT;
  _eRslt,
  _eState     : E_PROGRESS;
  _stMoveData : ST_MOVE_DATA; // dyn constraints for _MoverItf[i].Halt(Execute, stMoveData)
END_VAR
//-----------------------------------------------------------------------------
IF NOT Execute 
THEN 
	_eState                       := E_PROGRESS.PROGRESS_INIT; 
END_IF 
//-----------------------------------------------------------------------------
IF NOT Check() 
THEN 
	MoverHaltAll                  := E_PROGRESS.PROGRESS_ERROR; 
	RETURN; 
END_IF
//-----------------------------------------------------------------------------
//-----------------------------------------------------------------------------
CASE _eState
OF
  E_PROGRESS.PROGRESS_INIT:
    IF Execute
    THEN
      _nErrorId                 := 0;
      _nMover                   := 1;

      _eState                   := E_PROGRESS.PROGRESS_BUSY;
    END_IF
END_CASE
//-----------------------------------------------------------------------------
//-----------------------------------------------------------------------------
CASE _eState
OF
  E_PROGRESS.PROGRESS_BUSY:
    _eState                     := E_PROGRESS.PROGRESS_PREPARE;
    _stMoveData.rAcc            := _StationStart.rAccDec;
    _stMoveData.rGap            := _MoverLastGap[_nMover];

    IF NOT (_GroupInfo.AxisCount = MAX_MOVER)
    THEN
      _eRslt                    := _MoverItf[_nMover].Halt(FALSE, _stMoveData);
    ELSE
      _eRslt                    := _MoverItf[_nMover].HaltCa(FALSE, _stMoveData);
    END_IF
END_CASE
//-----------------------------------------------------------------------------
//-----------------------------------------------------------------------------
CASE _eState
OF
  E_PROGRESS.PROGRESS_PREPARE:
    IF NOT (_GroupInfo.AxisCount = MAX_MOVER)
    THEN
      _eRslt                    := _MoverItf[_nMover].Halt(TRUE, _stMoveData);
    ELSE
      _eRslt                    := _MoverItf[_nMover].HaltCa(TRUE, _stMoveData);
    END_IF

    IF (_eRslt = E_PROGRESS.PROGRESS_ERROR)
    THEN
      _eState                   := E_PROGRESS.PROGRESS_WORKING; // reset error on purpose, since we have to come back and get everybody in standstill
      _eRslt                    := _MoverItf[_nMover].Reset(FALSE);
      _nErrorId                 := _MoverInfo[_nMover].nErrorId; 

    ELSIF (_eRslt = E_PROGRESS.PROGRESS_DONE)
    THEN
      _eState                   := E_PROGRESS.PROGRESS_STARTUP;
    END_IF
END_CASE
//-----------------------------------------------------------------------------
//-----------------------------------------------------------------------------
CASE _eState
OF
  E_PROGRESS.PROGRESS_STARTUP:
    _eState                     := E_PROGRESS.PROGRESS_CHECK;

    IF NOT (_GroupInfo.AxisCount = MAX_MOVER)
    THEN
      _eRslt                    := _MoverItf[_nMover].Halt(FALSE, _stMoveData);
    ELSE
      _eRslt                    := _MoverItf[_nMover].HaltCa(FALSE, _stMoveData);
    END_IF

END_CASE
//-----------------------------------------------------------------------------
//-----------------------------------------------------------------------------
CASE _eState
OF
  E_PROGRESS.PROGRESS_CHECK:
    IF (_nMover > MAX_MOVER-1)
    THEN
      _eState                   := E_PROGRESS.PROGRESS_OCCUPIED;
    ELSE
      _nMover                   := _nMover + 1;
      _eState                   := E_PROGRESS.PROGRESS_BUSY;
    END_IF
END_CASE
//-----------------------------------------------------------------------------
//-----------------------------------------------------------------------------
CASE _eState
OF
  E_PROGRESS.PROGRESS_OCCUPIED:
    IF (_GroupInfo.AllAxesStanding)
    THEN
      _eState                   := E_PROGRESS.PROGRESS_DONE;

      IF (_eMessageLevel = E_MessageType.eMessageVerbose)
      THEN
        _stMsg.eType            := E_MessageType.eMessageVerbose;
        _stMsg.eSubdevice       := e_Subdevice.TransportUnit_General;
        _stMsg.iErrorNumber     := 0;
        _stMsg.sText            := concat( 'State: ', TO_STRING(THIS^._eState));
        _stMsg.sText            := concat(_stMsg.sText, ': ');
        _stMsg.sText            := concat(_stMsg.sText, TO_STRING(_eState));
        f_MessageSet(_stMsg);
      END_IF
    ELSE
      _nMover                   := 1;
      _eState                   := E_PROGRESS.PROGRESS_BUSY;
    END_IF
END_CASE
//-----------------------------------------------------------------------------
//-----------------------------------------------------------------------------
CASE _eState
OF
  E_PROGRESS.PROGRESS_WORKING:
    _eRslt                      := _MoverItf[_nMover].Reset(TRUE);

    IF (_eRslt = E_PROGRESS.PROGRESS_ERROR)
    THEN
      _eRslt                    := _MoverItf[_nMover].Reset(FALSE);
      _nErrorId                 := _MoverInfo[_nMover].nErrorId; 

    ELSIF (_eRslt = E_PROGRESS.PROGRESS_DONE)
    THEN
      _eState                   := E_PROGRESS.PROGRESS_BUSY;
      _eRslt                    := _MoverItf[_nMover].Reset(FALSE);
    END_IF
END_CASE
//-----------------------------------------------------------------------------
//-----------------------------------------------------------------------------

MoverHaltAll                    := _eState;
END_METHOD

PROPERTY MoverInfo : REFERENCE TO ARRAY[1..MAX_MOVER] OF ST_MOVER_INFO
SET
_MoverInfo REF= MoverInfo;
END_SET
END_PROPERTY

PROPERTY MoverItf : reference TO ARRAY[1..MAX_MOVER] OF I_XtsTransport_Mover
SET
_MoverItf REF= MoverItf;
END_SET
END_PROPERTY

PROPERTY MoverLastGap : REFERENCE to ARRAY[1..MAX_MOVER] of LREAL
SET
_MoverLastGap REF= MoverLastGap;
END_SET
END_PROPERTY

PROPERTY MoverLastPosition : REFERENCE to ARRAY[1..MAX_MOVER] of LREAL
SET
_MoverLastPosition REF= MoverLastPosition;
END_SET
END_PROPERTY

METHOD MoverStopAll : e_progress
VAR_INPUT
  Execute     : BOOL;
END_VAR
VAR_INST
  _nMover     : UINT;
  _nErrorId   : UDINT;
  _eRslt,
  _eState     : E_PROGRESS;
  _stMoveData : ST_MOVE_DATA; // dyn constraints for _MoverItf[i].Halt(Execute, stMoveData)
END_VAR
//-----------------------------------------------------------------------------
IF NOT Execute 
THEN 
	_eState                       := E_PROGRESS.PROGRESS_INIT; 
END_IF 
//-----------------------------------------------------------------------------
IF NOT Check() 
THEN 
	MoverStopAll                  := E_PROGRESS.PROGRESS_ERROR; 
	RETURN; 
END_IF
//-----------------------------------------------------------------------------
//-----------------------------------------------------------------------------
CASE _eState
OF
  E_PROGRESS.PROGRESS_INIT:
    IF Execute
    THEN
      _nErrorId                 := 0;
      _nMover                   := 1;

      _eState                   := E_PROGRESS.PROGRESS_BUSY;
    END_IF
END_CASE
//-----------------------------------------------------------------------------
//-----------------------------------------------------------------------------
CASE _eState
OF
  E_PROGRESS.PROGRESS_BUSY:
    _eState                     := E_PROGRESS.PROGRESS_PREPARE;
    _stMoveData.rAcc            := _StationStart.rAccDec;
    _stMoveData.rGap            := _MoverLastGap[_nMover];

    _eRslt                      := _MoverItf[_nMover].Stop(FALSE, _stMoveData);
END_CASE
//-----------------------------------------------------------------------------
//-----------------------------------------------------------------------------
CASE _eState
OF
  E_PROGRESS.PROGRESS_PREPARE:
    _eRslt                      := _MoverItf[_nMover].Stop(TRUE, _stMoveData);

    IF (_eRslt = E_PROGRESS.PROGRESS_ERROR)
    THEN
      _eState                   := E_PROGRESS.PROGRESS_WORKING; // reset error on purpose, since we have to come back and get everybody in standstill
      _eRslt                    := _MoverItf[_nMover].Reset(FALSE);
      _nErrorId                 := _MoverInfo[_nMover].nErrorId; 

    ELSIF (_eRslt = E_PROGRESS.PROGRESS_DONE)
    THEN
      _eState                   := E_PROGRESS.PROGRESS_STARTUP;
    END_IF
END_CASE
//-----------------------------------------------------------------------------
//-----------------------------------------------------------------------------
CASE _eState
OF
  E_PROGRESS.PROGRESS_STARTUP:
    _eState                     := E_PROGRESS.PROGRESS_CHECK;
    _eRslt                      := _MoverItf[_nMover].Halt(FALSE, _stMoveData);
END_CASE
//-----------------------------------------------------------------------------
//-----------------------------------------------------------------------------
CASE _eState
OF
  E_PROGRESS.PROGRESS_CHECK:
    IF (_nMover > MAX_MOVER-1)
    THEN
      _eState                   := E_PROGRESS.PROGRESS_OCCUPIED;
    ELSE
      _nMover                   := _nMover + 1;
      _eState                   := E_PROGRESS.PROGRESS_BUSY;
    END_IF
END_CASE
//-----------------------------------------------------------------------------
//-----------------------------------------------------------------------------
CASE _eState
OF
  E_PROGRESS.PROGRESS_OCCUPIED:
    IF (_GroupInfo.AllAxesStanding)
    THEN
      _eState                   := E_PROGRESS.PROGRESS_DONE;

      IF (_eMessageLevel = E_MessageType.eMessageVerbose)
      THEN
        _stMsg.eType            := E_MessageType.eMessageVerbose;
        _stMsg.eSubdevice       := e_Subdevice.TransportUnit_General;
        _stMsg.iErrorNumber     := 0;
        _stMsg.sText            := concat( 'State: ', TO_STRING(THIS^._eState));
        _stMsg.sText            := concat(_stMsg.sText, ': ');
        _stMsg.sText            := concat(_stMsg.sText, TO_STRING(_eState));
        f_MessageSet(_stMsg);
      END_IF
    ELSE
      _nMover                   := 1;
      _eState                   := E_PROGRESS.PROGRESS_BUSY;
    END_IF
END_CASE
//-----------------------------------------------------------------------------
//-----------------------------------------------------------------------------
CASE _eState
OF
  E_PROGRESS.PROGRESS_WORKING:
    _eRslt                      := _MoverItf[_nMover].Reset(TRUE);

    IF (_eRslt = E_PROGRESS.PROGRESS_ERROR)
    THEN
      _eRslt                    := _MoverItf[_nMover].Reset(FALSE);
      _nErrorId                 := _MoverInfo[_nMover].nErrorId; 

    ELSIF (_eRslt = E_PROGRESS.PROGRESS_DONE)
    THEN
      _eState                   := E_PROGRESS.PROGRESS_BUSY;
      _eRslt                    := _MoverItf[_nMover].Reset(FALSE);
    END_IF
END_CASE
//-----------------------------------------------------------------------------
//-----------------------------------------------------------------------------

MoverStopAll                    := _eState;
END_METHOD

PROPERTY State : REFERENCE TO ST_XTS_TRANSPORT_STATE
SET
_State ref= State;
END_SET
END_PROPERTY

PROPERTY StationControl : REFERENCE TO ARRAY[1..MAX_STATION]  OF ST_STATION_CTRL
SET
_StationControl REF= StationControl;
END_SET
END_PROPERTY

PROPERTY StationCtrlItf : REFERENCE TO ARRAY[1..MAX_STATION]  OF I_XtsTransport_Station;
SET
_ItfStationCtrl REF= StationCtrlItf;
END_SET
END_PROPERTY

PROPERTY StationListsItf : reference to ARRAY[1..MAX_STATION] OF I_Station_LinkedList
SET
_ItfStationList ref= StationListsItf;
END_SET
END_PROPERTY

METHOD StationsClearAll : E_PROGRESS
VAR_INPUT
  Execute     : BOOL;
END_VAR
VAR_INST
  _nStation,
  _nErrorId   : UDINT;
  _eJobReslt,
  _eState     : E_PROGRESS;
END_VAR
//-----------------------------------------------------------------------------
IF NOT Execute 
THEN 
	_eState                       := E_PROGRESS.PROGRESS_INIT; 
END_IF 
//-----------------------------------------------------------------------------
IF NOT Check() 
THEN 
	StationsClearAll              := E_PROGRESS.PROGRESS_ERROR; 
	RETURN; 
END_IF
//-----------------------------------------------------------------------------
//-----------------------------------------------------------------------------
CASE _eState
OF
  E_PROGRESS.PROGRESS_INIT:
    IF Execute
    THEN
      _nErrorId                 := 0;
      _nStation                 := 1;
      _eState                   := E_PROGRESS.PROGRESS_BUSY;
    END_IF
  //---------------------------------------------------------------------------
  //---------------------------------------------------------------------------
  E_PROGRESS.PROGRESS_BUSY:
    _eJobReslt                  := _ItfStationCtrl[_nStation].Init();

    IF (_eJobReslt = E_PROGRESS.PROGRESS_ERROR)
    THEN
      _eState                   := E_PROGRESS.PROGRESS_ERROR;
      _nErrorId                 := 669;

    ELSIF (_eJobReslt = E_PROGRESS.PROGRESS_DONE)
    THEN
      _eState                   := E_PROGRESS.PROGRESS_WORKING;
    END_IF

  //---------------------------------------------------------------------------
  //---------------------------------------------------------------------------
  E_PROGRESS.PROGRESS_WORKING:
    IF (_nStation < MAX_STATION)
    THEN
      _nStation                 := _nStation + 1;
      _eState                   := E_PROGRESS.PROGRESS_BUSY;
    ELSE
      _eState                   := E_PROGRESS.PROGRESS_DONE;

      IF (_eMessageLevel = E_MessageType.eMessageVerbose)
      THEN
        _stMsg.eType            := E_MessageType.eMessageVerbose;
        _stMsg.eSubdevice       := e_Subdevice.TransportUnit_General;
        _stMsg.iErrorNumber     := 0;
        _stMsg.sText            := concat( 'State: ', TO_STRING(THIS^._eState));
        _stMsg.sText            := concat(_stMsg.sText, ': ');
        _stMsg.sText            := concat(_stMsg.sText, TO_STRING(_eState));
        f_MessageSet(_stMsg);
      END_IF
    END_IF
END_CASE
//-----------------------------------------------------------------------------
//-----------------------------------------------------------------------------

StationsClearAll                := _eState;
END_METHOD

PROPERTY StationStart : reference to ST_STATION_PARAMETER
SET
_StationStart REF= StationStart;
END_SET
END_PROPERTY

PROPERTY StationStartIndex : uint
GET
StationStartIndex := _nStartStation;
END_GET
SET
_nStartStation := StationStartIndex;
END_SET
END_PROPERTY

PROPERTY StationState : REFERENCE TO ARRAY[1..MAX_STATION]  OF ST_STATION_STATE
SET
_StationState REF= StationState;
END_SET
END_PROPERTY

METHOD Template : E_PROGRESS
VAR_INPUT
  Execute     : BOOL;
END_VAR
VAR_INST
  _nErrorId   : UDINT;
  _eState     : E_PROGRESS;
END_VAR
//-----------------------------------------------------------------------------
IF NOT Execute 
THEN 
	_eState                       := E_PROGRESS.PROGRESS_INIT; 
END_IF 
//-----------------------------------------------------------------------------
IF NOT Check() 
THEN 
	Template_1                    := E_PROGRESS.PROGRESS_ERROR; 
	RETURN; 
END_IF
//-----------------------------------------------------------------------------
//-----------------------------------------------------------------------------
CASE _eState
OF
  E_PROGRESS.PROGRESS_INIT:
    IF Execute
    THEN
      _nErrorId                 := 0;

      _eState                   := E_PROGRESS.PROGRESS_BUSY;
    END_IF
END_CASE
//-----------------------------------------------------------------------------
//-----------------------------------------------------------------------------
CASE _eState
OF
  E_PROGRESS.PROGRESS_BUSY:
    _eState                     := E_PROGRESS.PROGRESS_PREPARE;
END_CASE
//-----------------------------------------------------------------------------
//-----------------------------------------------------------------------------
CASE _eState
OF
  E_PROGRESS.PROGRESS_PREPARE:

    IF (.Error)
    THEN
      _eState                   := E_PROGRESS.PROGRESS_ERROR;
      _nErrorId                 := 


    ELSIF (.Done)
    THEN
      _eState                   := E_PROGRESS.;

    END_IF
END_CASE
//-----------------------------------------------------------------------------
//-----------------------------------------------------------------------------

Template_1                      := _eState;
END_METHOD

METHOD TransportRestart : e_progress // movers must already to be error free, enabled and added to CA Group
VAR_INPUT
  Execute         : BOOL;
END_VAR
VAR_INST
  _StnState       : ST_STATION_STATE;

  _nStation,
  _nMover         : UINT;

  _nErrorId       : UDINT;

  _eRslt,
  _eState         : E_PROGRESS;
  
  _stMsg          : ST_Message;
  _stMoveData     : ST_MOVE_DATA;
END_VAR
//-----------------------------------------------------------------------------
IF NOT Execute 
THEN 
	_eState                       := E_PROGRESS.PROGRESS_INIT; 
END_IF 
//-----------------------------------------------------------------------------
IF NOT Check() 
THEN 
	TransportRestart              := E_PROGRESS.PROGRESS_ERROR; 
	RETURN; 
END_IF
//-----------------------------------------------------------------------------
//-----------------------------------------------------------------------------
CASE _eState
OF
  E_PROGRESS.PROGRESS_INIT:
    IF Execute
    THEN
      _nErrorId                 := 0;

      _nStation                 :=
      _nMover                   := 1;

      IF (_GroupInfo.AxisCountEnabled = MAX_MOVER)
      THEN
        _eState                 := E_PROGRESS.PROGRESS_BUSY;
      ELSE
        _eState                 := E_PROGRESS.PROGRESS_ERROR;

        _stMsg.eType            := E_MessageType.eMessageError;
        _stMsg.eSubdevice       := e_Subdevice.TransportUnit_Restart;
        _stMsg.iErrorNumber     := _GroupInfo.AxisCountEnabled;
        _stMsg.sText            := TO_STRING(_eState);
        _stMsg.sText            := concat(_stMsg.sText, ': _GroupInfo.AxisCountEnabled <> MAX_MOVER');
        f_MessageSet(_stMsg);
      END_IF
    END_IF
END_CASE
//-----------------------------------------------------------------------------
//-----------------------------------------------------------------------------
CASE _eState
OF
  E_PROGRESS.PROGRESS_BUSY:
    _StnState                   := _StationState[_nStation];

    CASE _StnState.eState
    OF
      E_STATION_STATE.STATION_ERROR_INFEED_ERROR:
        _StationControl[_nStation].eCmd := E_STATION_CTRL.STATION_MOVER_ENTER_RETRY;

      E_STATION_STATE.STATION_ERROR_OUTFEED_ERROR:
        _StationControl[_nStation].eCmd := E_STATION_CTRL.STATION_MOVER_GONE;

      E_STATION_STATE.STATION_ERROR_FATAL:
        _eState                 := E_PROGRESS.PROGRESS_ERROR;

        _stMsg.eType            := E_MessageType.eMessageError;
        _stMsg.eSubdevice       := e_Subdevice.TransportUnit_Restart;
        _stMsg.iErrorNumber     := _nStation;
        _stMsg.sText            := TO_STRING(_eState);
        _stMsg.sText            := concat(_stMsg.sText, ': _nStation STATION_ERROR_FATAL');
        f_MessageSet(_stMsg);

    ELSE
      _eState                   := E_PROGRESS.PROGRESS_PREPARE;  
    END_CASE
END_CASE
//-----------------------------------------------------------------------------
//-----------------------------------------------------------------------------
CASE _eState
OF
  E_PROGRESS.PROGRESS_PREPARE:
    IF (_nStation > MAX_STATION-1)
    THEN
      _eState                   := E_PROGRESS.PROGRESS_STARTUP;
    ELSE
      _nStation                 := _nStation + 1;
      _eState                   := E_PROGRESS.PROGRESS_BUSY;
    END_IF
END_CASE
//-----------------------------------------------------------------------------
//-----------------------------------------------------------------------------
CASE _eState
OF
  E_PROGRESS.PROGRESS_STARTUP:
    _stMoveData.rPos            := _MoverLastPosition[_nMover];
    _stMoveData.rGap            := _MoverLastGap     [_nMover];

    _stMoveData.rVelo           := _StationStart.rVelo;
    _stMoveData.rAcc            := _StationStart.rAccDec;
    _stMoveData.rJerk           := _StationStart.rJerk;

    _stMoveData.rDelta          :=   0.1;
    _stMoveData.rDistance       :=  -1.0;
    _stMoveData.rOverride       := 100.0;

    _eRslt                      := _MoverItf[_nMover].SendToAbsPosCa(FALSE, _stMoveData);

